// TIA Portal project "labE000120203ICA" (V15.1)

(* hardware
DEVICE "S7300/ET200M station_2"  S7-300 station
   slot 0: "Rail_0"  Rail  6ES7 390-1***0-0AA0
   slot 2: "PLC_Shaft"  CPU 314C-2 PN/DP  6ES7 314-6EH04-0AB0  V3.3
      slot 2: "PROFINET interface_1"  PN-IO
         slot 1: "Port_1"  Port
         slot 2: "Port_2"  Port
      slot 5: "DI 24/DO 16_1"  DI24/DO16
      slot 6: "AI 5/AO 2_1"  AI5/AO2
      slot 7: "Count_1"  Counter
      slot 8: "Positioning_1"  Positioning
DEVICE "HMI_Shaft"  KTP700 Basic PN
   slot 0: "HMI_Shaft"  KTP700 Basic PN  6AV2 123-2GB03-0AX0  15.1.0.0
   slot 1: "HMI_RT_2"  KTP700 Basic PN  6AV2 123-2GB03-0AX0  15.1.0.0
   slot 5: "HMI_Shaft.IE_CP_1"  PROFINET Interface  15.0.1.0
      slot 1: "PROFINET Interface_1"  PROFINET Interface
         slot 1: "Port_1"  Port
DEVICE "ET 200SP station_1"  ET 200SP-Station
   slot 0: "Rack_0"  Rack  6ES5 710-8MAx1
   slot 0: "IO device_1"  IM 155-6 PN/2 HF  6ES7 155-6AU01-0CN0  V4.2
   slot 1: "Server module_1"  Server module  6ES7 193-6PA00-0AA0  V1.1
      slot 1: "Server module_1"  Server module
   slot 127: "BA 2xRJ45"  BA 2xRJ45  6ES7 193-6AR00-0AA0  V0.0
      slot 1: "Port_1"  X1 P1 R  6ES7 193-6AR00-0AA0  V0.0
      slot 2: "Port_2"  X1 P2 R  6ES7 193-6AR00-0AA0  V0.0
DEVICE "S71500/ET200MP station_1"  S7-1500 station
   slot 0: "Rail_0"  Rack  6ES7 590-1***0-0AA0
   slot 1: "PLC_1"  CPU 1516-3 PN/DP  6ES7 516-3AN01-0AB0  V2.6
      slot 3: "CPU display_1"  6ES7591-1BA00-0AA0
*)

// ===== PLC "PLC_Shaft"  CPU 314C-2 PN/DP =====

TYPE "carousel"
   STRUCT
      carousel : Array[0..7] of Int;
   END_STRUCT;
END_TYPE

TYPE "Sequence"
VERSION : 0.1
   STRUCT
      actual : "step";
      old : "step";
      break : "step";
   END_STRUCT;
END_TYPE

TYPE "step"
VERSION : 0.1
   STRUCT
      "step" : Array[0..25] of Bool;
   END_STRUCT;
END_TYPE

TYPE "CTRL"
VERSION : 0.1
   STRUCT
      emergency_stop : Bool;
      trigger : Bool;
      trigger_flank : Bool;
      trigger_toggle : Bool;
      trigger_hulp : Bool;
      enable_step : Bool;
      auto : Bool;
      onestep : Bool;
      step_stop : Bool;
      step_break : Bool;
      toggle_hulp : Bool;
      break_on : Bool;
   END_STRUCT;
END_TYPE

TYPE "grafcet_data"
VERSION : 0.1
   STRUCT
      MyCTRL : "CTRL";
      Mygrafcet : "Sequence";
   END_STRUCT;
END_TYPE

DATA_BLOCK "Tafel_As_DB"   // DB1
{ S7_Optimized_Access := 'FALSE' }
VERSION : 0.1
// stored: InstanceOfName Tafel_As
"Tafel_As"
BEGIN
END_DATA_BLOCK

FUNCTION_BLOCK "Tafel_As"   // FB1, SCL
{ S7_Optimized_Access := 'FALSE' }
VERSION : 0.1
   VAR_INPUT
      sensorA0 : Bool;
      sensorA1 : Bool;
      sensorB0 : Bool;
      sensorB1 : Bool;
      sensorC0 : Bool;
      sensorC1 : Bool;
      sensorD0 : Bool;
      sensorD1 : Bool;
      sensorF1 : Bool;
      sensorG0 : Bool;
      sensorG1 : Bool;
      sensorV1 : Bool;
      sensorV2 : Bool;
      sensorDm : Bool;
      sensorDp : Bool;
      sensorJ0 : Bool;
   END_VAR
   VAR_OUTPUT
      "CilA+" : Bool;
      "CilB+" : Bool;
      "CilC+" : Bool;
      "CilC-" : Bool;
      "CilD+" : Bool;
      "CilE+" : Bool;
      "CilF+" : Bool;
      "CilG+" : Bool;
      "CilH+" : Bool;
      "CilI+" : Bool;
      "CilK+" : Bool;
      "CilJ+" : Bool;
      "ZV1+" : Bool;
      "ZV2+" : Bool;
   END_VAR
   VAR
      "cilinderA+" : "cilinder";
      "cilinderB+" : "cilinder";
      "cilinderC+" : "cilinder";
      "cilinderC-" : "cilinder";
      "cilinderD+" : "cilinder";
      "cilinderE+" : "cilinder";
      "cilinderF+" : "cilinder";
      "cilinderG+" : "cilinder";
      "cilinderH+" : "cilinder";
      "cilinderI+" : "cilinder";
      "cilinderK+" : "cilinder";
      "cilinderJ+" : "cilinder";
      "zuigerV1+" : "cilinder";
      "zuigerV2+" : "cilinder";
      seq_as_einde_invoer : "grafcet_data";
      seq_as_draaien_invoer : "grafcet_data";
      seq_sorteringsarm_invoer : "grafcet_data";
      seq_detectiesensoren_invoer : "grafcet_data";
      seq_carousel_invoer : "grafcet_data";
      timer300ms : TON;
   END_VAR
BEGIN
   REGION Aanmaken grafcets
       // Statement section REGION
       "ctrl_seq"(size := 10,
                  sequences := #seq_as_einde_invoer);

       "ctrl_seq"(size := 10,
                  sequences := #seq_as_draaien_invoer);

       "ctrl_seq"(size := 10,
                  sequences := #seq_sorteringsarm_invoer);

       "ctrl_seq"(size := 10,
                  sequences := #seq_detectiesensoren_invoer);

       "ctrl_seq"(size := 10,
                  sequences := #seq_carousel_invoer);
   END_REGION


   REGION Stappen grafcet as plaatsen op lager
       // Statement section REGION
       "Seq1-->1"(actualstep := 1,
                  nextstep := 2,
                  condition := #sensorB0,
                  Sequence := #seq_as_einde_invoer);

       "Seq1-->1"(actualstep := 2,
                  nextstep := 3,
                  condition := #sensorA0,
                  Sequence := #seq_as_einde_invoer);

       "Seq1-->1"(actualstep := 3,
                  nextstep := 4,
                  condition := #sensorA1,
                  Sequence := #seq_as_einde_invoer);

       "Seq1-->1"(actualstep := 4,
                  nextstep := 5,
                  condition := #sensorV1,
                  Sequence := #seq_as_einde_invoer);

       "Seq1-->1"(actualstep := 5,
                  nextstep := 6,
                  condition := #sensorA0,
                  Sequence := #seq_as_einde_invoer);

       "Seq1-->1"(actualstep := 6,
                  nextstep := 7,
                  condition := #sensorB1,
                  Sequence := #seq_as_einde_invoer);

       "Seq1-->1"(actualstep := 7,
                  nextstep := 8,
                  condition := #sensorA1,
                  Sequence := #seq_as_einde_invoer);

       "Seq1-->1"(actualstep := 8,
                  nextstep := 9,
                  condition := #timer300ms.Q,
                  Sequence := #seq_as_einde_invoer);

       "Seq1-->1"(actualstep := 9,
                  nextstep := 1,
                  condition := #sensorA0,
                  Sequence := #seq_as_einde_invoer);
   END_REGION

   REGION Stappen grafcet as draaien
       // Statement section REGION
       "Seq1-->1"(actualstep := 1,
                  nextstep := 2,
                  condition := #sensorG0,
                  Sequence := #seq_as_draaien_invoer);

       "Seq1-->1"(actualstep := 2,
                  nextstep := 3,
                  condition := #sensorG1,
                  Sequence := #seq_as_draaien_invoer);

       "Seq1-->1"(actualstep := 3,
                  nextstep := 4,
                  condition := #timer300ms.Q,
                  Sequence := #seq_as_draaien_invoer);

       "Seq1-->1"(actualstep := 4,
                  nextstep := 5,
                  condition := #sensorG0,
                  Sequence := #seq_as_draaien_invoer);

       "Seq1-->1"(actualstep := 5,
                  nextstep := 6,
                  condition := #timer300ms.Q,
                  Sequence := #seq_as_draaien_invoer);

       "Seq1-->1"(actualstep := 6,
                  nextstep := 7,
                  condition := #sensorG1,
                  Sequence := #seq_as_draaien_invoer);

       "Seq1-->1"(actualstep := 7,
                  nextstep := 8,
                  condition := #sensorG1,
                  Sequence := #seq_as_draaien_invoer);

       "Seq1-->1"(actualstep := 8,
                  nextstep := 1,
                  condition := #timer300ms.Q,
                  Sequence := #seq_as_draaien_invoer);
   END_REGION

   REGION Stappen grafset sorteringsarm
       // Statement section REGION
       "Seq1-->1"(actualstep := 1,
                  nextstep := 2,
                  condition := #sensorC0,
                  Sequence := #seq_sorteringsarm_invoer);

       "Seq1-->1"(actualstep := 2,
                  nextstep := 3,
                  condition := #sensorC1,
                  Sequence := #seq_sorteringsarm_invoer);

       "Seq1-->1"(actualstep := 3,
                  nextstep := 4,
                  condition := #sensorD1,
                  Sequence := #seq_sorteringsarm_invoer);

       "Seq1-->1"(actualstep := 4,
                  nextstep := 5,
                  condition := #sensorV2,
                  Sequence := #seq_sorteringsarm_invoer);

       "Seq1-->1"(actualstep := 5,
                  nextstep := 1,
                  condition := #sensorD0,
                  Sequence := #seq_sorteringsarm_invoer);
   END_REGION

   REGION Stappen grafcet carousel
       // Statement section REGION
       "Seq1-->1"(actualstep:=1,
                  nextstep:=2,
                  condition:=#sensorJ0,
                  Sequence:=#seq_carousel_invoer);

       "Seq1-->1"(actualstep:=2,
                  nextstep:=3,
                  condition:=#seq_as_draaien_invoer.Mygrafcet.actual.step[8] AND #seq_as_einde_invoer.Mygrafcet.actual.step[9] AND #seq_sorteringsarm_invoer.Mygrafcet.actual.step[5],
                  Sequence:=#seq_carousel_invoer);

       "Seq1-->1"(actualstep:=3,
                  nextstep:=4,
                  condition:=#timer300ms.Q,
                  Sequence:=#seq_carousel_invoer);

       "Seq1-->1"(actualstep:=4,
                  nextstep:=5,
                  condition:=#timer300ms.Q AND #sensorJ0 = FALSE,
                  Sequence:=#seq_carousel_invoer);

       "Seq1-->1"(actualstep:=5,
                  nextstep:=1,
                  condition:=#timer300ms.Q,
                  Sequence:=#seq_carousel_invoer);

   END_REGION



   REGION Uitgangen as draaien
       // Statement section REGION
       #"cilinderH+"(manueelinschuiven := false,
                     manueeluitschuiven := false,
                     AutomatischUitschuiven := #seq_as_draaien_invoer.Mygrafcet.actual.step[4] OR #seq_as_einde_invoer.Mygrafcet.actual.step[5] OR #seq_as_einde_invoer.Mygrafcet.actual.step[6] OR #seq_as_einde_invoer.Mygrafcet.actual.step[7],
                     ManAuto := false,
                     "IL uitschuiven" := false,
                     "IL inschuiven" := false,
                     "Eindeloop In" := false,
                     "Eindeloop Uit" := false,
                     "Reset Foutmelding" := false,
                     TeachMode := false,
                     MargeLooptijden := T#0ms,
                     "Max Aantal slagen" := 0,
                     "Reset Onderhoud" := false,
                     Noodstop := false,
                     AansturingMono =>#"CilH+");

       #"cilinderG+"(manueelinschuiven := false,
                     manueeluitschuiven := false,
                     AutomatischUitschuiven:=#seq_as_draaien_invoer.Mygrafcet.actual.step[1] OR #seq_as_draaien_invoer.Mygrafcet.actual.step[2] OR #seq_as_draaien_invoer.Mygrafcet.actual.step[5] OR #seq_as_draaien_invoer.Mygrafcet.actual.step[6],
                     ManAuto := false,
                     "IL uitschuiven" := false,
                     "IL inschuiven" := false,
                     "Eindeloop In" := false,
                     "Eindeloop Uit" := false,
                     "Reset Foutmelding" := false,
                     TeachMode := false,
                     MargeLooptijden := T#0ms,
                     "Max Aantal slagen" := 0,
                     "Reset Onderhoud" := false,
                     Noodstop := false,
                     AansturingMono=>#"CilG+");

       #"cilinderI+"(manueelinschuiven := false,
                     manueeluitschuiven := false,
                     AutomatischUitschuiven:=#seq_as_draaien_invoer.Mygrafcet.actual.step[2] OR #seq_as_draaien_invoer.Mygrafcet.actual.step[3] OR #seq_as_draaien_invoer.Mygrafcet.actual.step[4] OR #seq_as_draaien_invoer.Mygrafcet.actual.step[5],
                     ManAuto := false,
                     "IL uitschuiven" := false,
                     "IL inschuiven" := false,
                     "Eindeloop In" := false,
                     "Eindeloop Uit" := false,
                     "Reset Foutmelding" := false,
                     TeachMode := false,
                     MargeLooptijden := T#0ms,
                     "Max Aantal slagen" := 0,
                     "Reset Onderhoud" := false,
                     Noodstop := false,
                     AansturingMono=>#"CilI+");

   END_REGION

   REGION Uitgangen as plaatsen op lager
       // Statement section REGION
       #"cilinderA+"(manueelinschuiven := false,
                     manueeluitschuiven := false,
                     AutomatischUitschuiven := #seq_as_einde_invoer.Mygrafcet.actual.step[2] OR #seq_as_einde_invoer.Mygrafcet.actual.step[3] OR #seq_as_einde_invoer.Mygrafcet.actual.step[6] OR #seq_as_einde_invoer.Mygrafcet.actual.step[7],
                     ManAuto := false,
                     "IL uitschuiven" := #sensorA0,
                     "IL inschuiven" := #sensorA1,
                     "Eindeloop In" := false,
                     "Eindeloop Uit" := false,
                     "Reset Foutmelding" := false,
                     TeachMode := false,
                     MargeLooptijden := T#0ms,
                     "Max Aantal slagen" := 0,
                     "Reset Onderhoud" := false,
                     Noodstop := false,
                     AansturingMono => #"CilA+");


       #"cilinderB+"(manueelinschuiven := false,
                     manueeluitschuiven := false,
                     AutomatischUitschuiven := #seq_as_einde_invoer.Mygrafcet.actual.step[5] OR #seq_as_einde_invoer.Mygrafcet.actual.step[6] OR #seq_as_einde_invoer.Mygrafcet.actual.step[7] OR #seq_as_einde_invoer.Mygrafcet.actual.step[8],
                     ManAuto := false,
                     "IL uitschuiven" := #sensorB0,
                     "IL inschuiven" := #sensorB1,
                     "Eindeloop In" := false,
                     "Eindeloop Uit" := false,
                     "Reset Foutmelding" := false,
                     TeachMode := false,
                     MargeLooptijden := T#0ms,
                     "Max Aantal slagen" := 0,
                     "Reset Onderhoud" := false,
                     Noodstop := false,
                     AansturingMono => #"CilB+");


       #"zuigerV1+"(manueelinschuiven := false,
                    manueeluitschuiven := false,
                    AutomatischUitschuiven:=#seq_as_einde_invoer.Mygrafcet.actual.step[3] OR #seq_as_einde_invoer.Mygrafcet.actual.step[4] OR #seq_as_einde_invoer.Mygrafcet.actual.step[5] OR #seq_as_einde_invoer.Mygrafcet.actual.step[6],
                    ManAuto := false,
                    "IL uitschuiven" := false,
                    "IL inschuiven" := false,
                    "Eindeloop In" := false,
                    "Eindeloop Uit" := false,
                    "Reset Foutmelding" := false,
                    TeachMode := false,
                    MargeLooptijden := T#0ms,
                    "Max Aantal slagen" := 0,
                    "Reset Onderhoud" := false,
                    Noodstop := false,
                    AansturingMono=>#"ZV1+");
   END_REGION

   REGION Uitgangen sorteringsarm
       // Statement section REGION
       #"cilinderC+"(manueelinschuiven := false,
                     manueeluitschuiven := false,
                     AutomatischUitschuiven:=#seq_sorteringsarm_invoer.Mygrafcet.actual.step[1],
                     ManAuto := false,
                     "IL uitschuiven" := false,
                     "IL inschuiven" := false,
                     "Eindeloop In" := false,
                     "Eindeloop Uit" := false,
                     "Reset Foutmelding" := false,
                     TeachMode := false,
                     MargeLooptijden := T#0ms,
                     "Max Aantal slagen" := 0,
                     "Reset Onderhoud" := false,
                     Noodstop := false,
                     AansturingMono=>#"CilC+");

       #"cilinderC-"(manueelinschuiven := false,
                     manueeluitschuiven := false,
                     AutomatischUitschuiven:=#seq_sorteringsarm_invoer.Mygrafcet.actual.step[5],
                     ManAuto := false,
                     "IL uitschuiven" := false,
                     "IL inschuiven" := false,
                     "Eindeloop In" := false,
                     "Eindeloop Uit" := false,
                     "Reset Foutmelding" := false,
                     TeachMode := false,
                     MargeLooptijden := T#0ms,
                     "Max Aantal slagen" := 0,
                     "Reset Onderhoud" := false,
                     Noodstop := false,
                     AansturingMono=>#"CilC-");

       #"cilinderD+"(manueelinschuiven := false,
                     manueeluitschuiven := false,
                     AutomatischUitschuiven:=#seq_sorteringsarm_invoer.Mygrafcet.actual.step[2] OR #seq_sorteringsarm_invoer.Mygrafcet.actual.step[3],
                     ManAuto := false,
                     "IL uitschuiven" := false,
                     "IL inschuiven" := false,
                     "Eindeloop In" := false,
                     "Eindeloop Uit" := false,
                     "Reset Foutmelding" := false,
                     TeachMode := false,
                     MargeLooptijden := T#0ms,
                     "Max Aantal slagen" := 0,
                     "Reset Onderhoud" := false,
                     Noodstop := false,
                     AansturingMono=>#"CilD+");

       #"zuigerV2+"(manueelinschuiven := false,
                    manueeluitschuiven := false,
                    AutomatischUitschuiven:=#seq_sorteringsarm_invoer.Mygrafcet.actual.step[3] OR #seq_sorteringsarm_invoer.Mygrafcet.actual.step[4] OR #seq_sorteringsarm_invoer.Mygrafcet.actual.step[5],
                    ManAuto := false,
                    "IL uitschuiven" := false,
                    "IL inschuiven" := false,
                    "Eindeloop In" := false,
                    "Eindeloop Uit" := false,
                    "Reset Foutmelding" := false,
                    TeachMode := false,
                    MargeLooptijden := T#0ms,
                    "Max Aantal slagen" := 0,
                    "Reset Onderhoud" := false,
                    Noodstop := false,
                    AansturingMono=>#"ZV2+");

   END_REGION

   REGION Uitgang carousel
       // Statement section REGION
       #"cilinderK+"(manueelinschuiven := false,
                     manueeluitschuiven := false,
                     AutomatischUitschuiven:=#seq_carousel_invoer.Mygrafcet.actual.step[2] OR #seq_carousel_invoer.Mygrafcet.actual.step[3],
                     ManAuto := false,
                     "IL uitschuiven" := false,
                     "IL inschuiven" := false,
                     "Eindeloop In" := false,
                     "Eindeloop Uit" := false,
                     "Reset Foutmelding" := false,
                     TeachMode := false,
                     MargeLooptijden := T#0ms,
                     "Max Aantal slagen" := 0,
                     "Reset Onderhoud" := false,
                     Noodstop := false,
                     AansturingMono=>#"CilK+");

       #"cilinderJ+"(manueelinschuiven := false,
                     manueeluitschuiven := false,
                     AutomatischUitschuiven:=#seq_carousel_invoer.Mygrafcet.actual.step[3] OR #seq_carousel_invoer.Mygrafcet.actual.step[4],
                     ManAuto := false,
                     "IL uitschuiven" := false,
                     "IL inschuiven" := false,
                     "Eindeloop In" := false,
                     "Eindeloop Uit" := false,
                     "Reset Foutmelding" := false,
                     TeachMode := false,
                     MargeLooptijden := T#0ms,
                     "Max Aantal slagen" := 0,
                     "Reset Onderhoud" := false,
                     Noodstop := false,
                     AansturingMono=>#"CilJ+");

   END_REGION



   #timer300ms(IN := #seq_carousel_invoer.Mygrafcet.actual.step[2] OR #seq_carousel_invoer.Mygrafcet.actual.step[3] OR #seq_carousel_invoer.Mygrafcet.actual.step[4] OR #seq_as_einde_invoer.Mygrafcet.actual.step[7] OR #seq_as_draaien_invoer.Mygrafcet.actual.step[3] OR #seq_as_draaien_invoer.Mygrafcet.actual.step[5] OR #seq_as_draaien_invoer.Mygrafcet.actual.step[7],
               PT := t#300ms);
END_FUNCTION_BLOCK

ORGANIZATION_BLOCK "Main"   // OB1, LAD
TITLE = "Main Program Sweep (Cycle)"
{ S7_Optimized_Access := 'FALSE' }
VERSION : 0.1
   VAR_TEMP
      OB1_EV_CLASS : Byte;   // Bits 0-3 = 1 (Coming event), Bits 4-7 = 1 (Event class 1)
      OB1_SCAN_1 : Byte;   // 1 (Cold restart scan 1 of OB 1), 3 (Scan 2-n of OB 1)
      OB1_PRIORITY : Byte;   // Priority of OB Execution
      OB1_OB_NUMBR : Byte;   // 1 (Organization block 1, OB1)
      OB1_RESERVED_1 : Byte;   // Reserved for system
      OB1_RESERVED_2 : Byte;   // Reserved for system
      OB1_PREV_CYCLE : Int;   // Cycle time of previous OB1 scan (milliseconds)
      OB1_MIN_CYCLE : Int;   // Minimum cycle time of OB1 (milliseconds)
      OB1_MAX_CYCLE : Int;   // Maximum cycle time of OB1 (milliseconds)
      OB1_DATE_TIME : Date_And_Time;   // Date and time OB1 started
   END_VAR
BEGIN

REGION Network 1
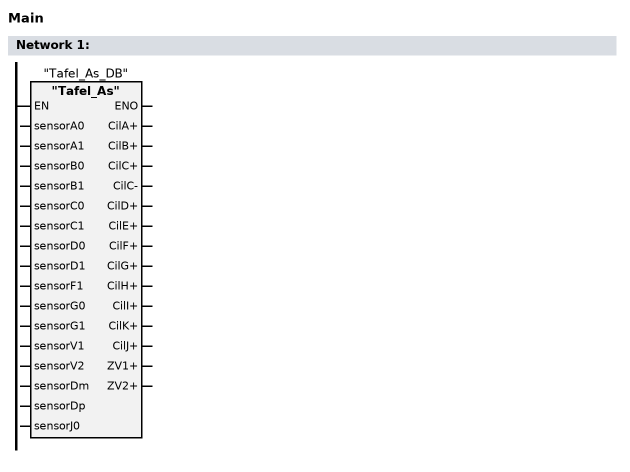
   RUNG wire#powerrail
      "Tafel_As_DB"(sensorA0 :=, sensorA1 :=, sensorB0 :=, sensorB1 :=, sensorC0 :=, sensorC1 :=, sensorD0 :=, sensorD1 :=, sensorF1 :=, sensorG0 :=, sensorG1 :=, sensorV1 :=, sensorV2 :=, sensorDm :=, sensorDp :=, sensorJ0 :=, "CilA+" =>, "CilB+" =>, "CilC+" =>, "CilC-" =>, "CilD+" =>, "CilE+" =>, "CilF+" =>, "CilG+" =>, "CilH+" =>, "CilI+" =>, "CilK+" =>, "CilJ+" =>, "ZV1+" =>, "ZV2+" =>)
   END_RUNG
   // the same network as SCL:
   "Tafel_As_DB"();   // "Tafel_As"
END_REGION
END_ORGANIZATION_BLOCK

ORGANIZATION_BLOCK "COMPLETE RESTART"   // OB100, SCL
TITLE = "Complete Restart"
{ S7_Optimized_Access := 'FALSE' }
VERSION : 0.1
   VAR_TEMP
      OB100_EV_CLASS : Byte;   // 16#13, Event class 1, Entering event state, Event logged in diagnostic buffer
      OB100_STRTUP : Byte;   // 16#81/82/83/84 Method of startup
      OB100_PRIORITY : Byte;   // Priority of OB Execution
      OB100_OB_NUMBR : Byte;   // 100 (Organization block 100, OB100)
      OB100_RESERVED_1 : Byte;   // Reserved for system
      OB100_RESERVED_2 : Byte;   // Reserved for system
      OB100_STOP : Word;   // Event that caused CPU to stop (16#4xxx)
      OB100_STRT_INFO : DWord;   // Information on how system started
      OB100_DATE_TIME : Date_And_Time;   // Date and time OB100 started
   END_VAR
BEGIN
   "initialisation"(number:=20,
                    Normal_sequence:="Mijn_Tafel_Lager".seq_invoer);
   "initialisation"(number := 20,
                    Normal_sequence := "Mijn_Tafel_Lager".seq_uitvoer);
END_ORGANIZATION_BLOCK

// folder: basisclasses

FUNCTION_BLOCK "cilinder"   // FB8, FBD
{ S7_Optimized_Access := 'FALSE' }
VERSION : 0.1
   VAR_INPUT
      manueelinschuiven : Bool;
      manueeluitschuiven : Bool;   // '1' betekent uitschuiven '0' inschuiven
      AutomatischUitschuiven : Bool;
      ManAuto : Bool;   // '1' betekent Manueel '0' Automatisch
      "IL uitschuiven" : Bool;   // '1' betekent vergrendeld
      "IL inschuiven" : Bool;   // '1' betekent vergrendeld
      "Eindeloop In" : Bool;
      "Eindeloop Uit" : Bool;
      "Reset Foutmelding" : Bool;
      TeachMode : Bool;   // '1' wanneer er tijden worden ingesteld
      MargeLooptijden : Time;   // marge instellen looptijdbewaking
      "Max Aantal slagen" : Int;   // Aantal slagen voor onderhoud
      "Reset Onderhoud" : Bool;
      Noodstop : Bool;   // '0' betekent noodstop actief
   END_VAR
   VAR_OUTPUT
      AansturingMono : Bool;
      AansturingAanBist : Bool;
      AansturingUitBist : Bool;
      "Alarm Looptijd" : Bool;   // Te lang om dicht of open te schuiven
      "Alarm Interlock" : Bool;   // poging om te bedienen bij aanwezige interlock
      "Alarm Noodstop" : Bool;
      "Alarm Eindeloop" : Bool;   // wanneer elektrisch probleem op eindelopen
      "Alarm Onderhoud" : Bool;
   END_VAR
   VAR
      grafcetssturing : Bool;
      "Referentie Looptijd Inschuiven" : Time;
      "Referentie Looptijd Uitschuiven" : Time;
      "Werkelijke Looptijd Inschuiven" : Time;
      "Werkelijke Looptijd Uitschuiven" : Time;
      "Werkelijke Aantal Slagen" : Int;
      OnderhoudTeller : CTD;
      SROnderhoud : Bool;
      SREindeloop : Bool;
      SRNoodstop : Bool;
      FlankManUit : Bool;
      FlankAutoUit : Bool;
      SRInterlock : Bool;
      FlankManIN : Bool;
      FlankAutoIN : Bool;
      TeachTimer : TON;
      FlankEindeUit : Bool;
      FlankEindeIn : Bool;
      RefTijdIn : Int;
      RefTijdUit : Int;
      WerkTijdIn : Int;
      WerkTijdUit : Int;
      SRLooptijd : Bool;
      FlankEindeUit1 : Bool;
      FlankEindeIn1 : Bool;
      eindeloopuitflank : Bool;
      eindeloopinflank : Bool;
      bewaaktijdeninschuiven : "bewaaktijden";
      bewaaktijdenuitschuif : "bewaaktijden";
      flankmanueelinschuiven : Bool;
      flankmanueeluitschuiven : Bool;
      movesetreset : Bool;
      PercentageSlagen : Real;
      Real_aantal : Real;
      Monosturing : Bool;
      BisturingAan : Bool;
      BisturingUit : Bool;
      FposAansturing : Bool;
      FnegAansturing : Bool;
      DINT_aantal : DInt;
   END_VAR
   VAR_TEMP
      ondergrensin : Int;
      bovengrensuit : Int;
      ondergrensuit : Int;
      vals : Bool;
      bovengrensin : Int;
   END_VAR
   VAR_TEMP   // added for the SCL form of the ladder/FBD networks
      _w1 : Bool;
      _w2 : Bool;
      _w3 : Bool;
      _w4 : Bool;
      _w5 : Bool;
   END_VAR
BEGIN

REGION Network 1: Onderhoud
   // Teller van de cilindir om na x aantal slagen onderhoud uit te voeren op de cilindir.
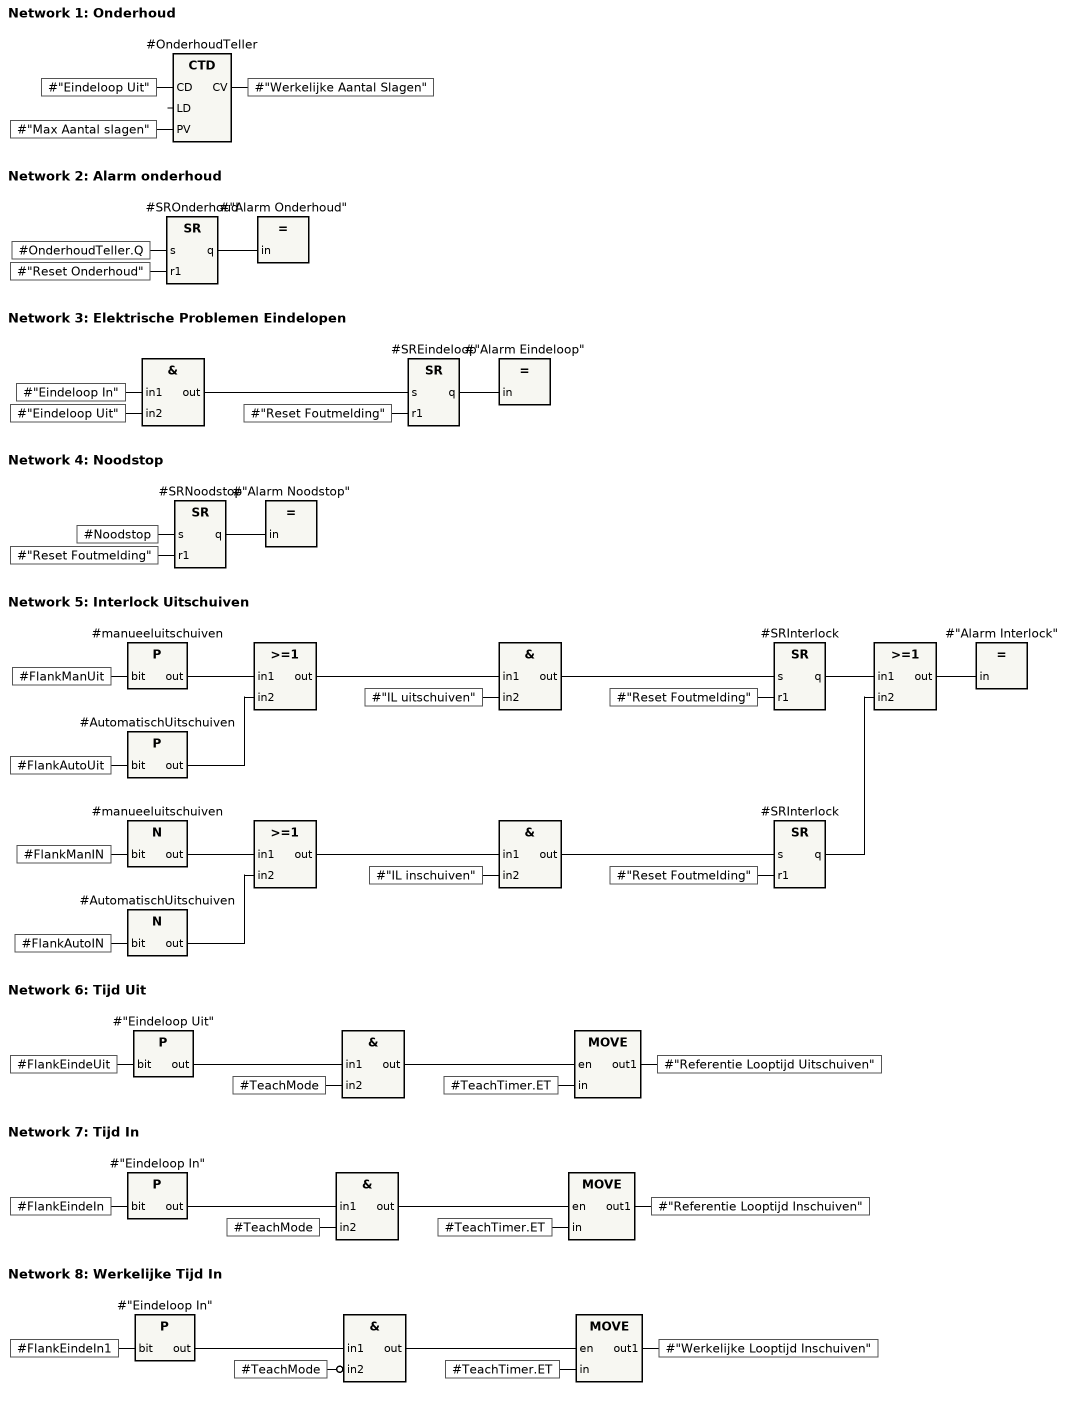
   #OnderhoudTeller.CTD(CD := #"Eindeloop Uit", PV := #"Max Aantal slagen", CV => #"Werkelijke Aantal Slagen");
END_REGION

REGION Network 2: Alarm onderhoud
   // Weergave van wanneer de teller zijn aantal slagen heeft bereikt, kan gereset worden
   IF #OnderhoudTeller.Q THEN
       #SROnderhoud := TRUE;   // SR flip-flop
   END_IF;
   IF #"Reset Onderhoud" THEN #SROnderhoud := FALSE; END_IF;
   #"Alarm Onderhoud" := #SROnderhoud;
END_REGION

REGION Network 3: Elektrische Problemen Eindelopen
   // Beide eindelopen mogen nooit beide aanliggen, dit is fysisch niet mogelijk en is dus een elektrisch probleem
   IF #"Eindeloop In" AND #"Eindeloop Uit" THEN
       #SREindeloop := TRUE;   // SR flip-flop
   END_IF;
   IF #"Reset Foutmelding" THEN #SREindeloop := FALSE; END_IF;
   #"Alarm Eindeloop" := #SREindeloop;
END_REGION

REGION Network 4: Noodstop
   // de fysishe noodstop is nc contact
   IF #Noodstop THEN
       #SRNoodstop := TRUE;   // SR flip-flop
   END_IF;
   IF #"Reset Foutmelding" THEN #SRNoodstop := FALSE; END_IF;
   #"Alarm Noodstop" := #SRNoodstop;
END_REGION

REGION Network 5: Interlock Uitschuiven
   // Alarm voor wanneer de cilindir wordt aangestuurd maar de interlock is actief.
   #_w1 := #manueeluitschuiven AND NOT #FlankManUit;   // rising edge of #manueeluitschuiven
   #FlankManUit := #manueeluitschuiven;
   #_w2 := #AutomatischUitschuiven AND NOT #FlankAutoUit;   // rising edge of #AutomatischUitschuiven
   #FlankAutoUit := #AutomatischUitschuiven;
   IF (#_w1 OR #_w2) AND #"IL uitschuiven" THEN
       #SRInterlock := TRUE;   // SR flip-flop
   END_IF;
   IF #"Reset Foutmelding" THEN #SRInterlock := FALSE; END_IF;
   #_w3 := NOT #manueeluitschuiven AND #FlankManIN;   // falling edge of #manueeluitschuiven
   #FlankManIN := #manueeluitschuiven;
   #_w4 := NOT #AutomatischUitschuiven AND #FlankAutoIN;   // falling edge of #AutomatischUitschuiven
   #FlankAutoIN := #AutomatischUitschuiven;
   #_w5 := #SRInterlock;
   IF (#_w3 OR #_w4) AND #"IL inschuiven" THEN
       #SRInterlock := TRUE;   // SR flip-flop
   END_IF;
   IF #"Reset Foutmelding" THEN #SRInterlock := FALSE; END_IF;
   #"Alarm Interlock" := #_w5 OR #SRInterlock;
END_REGION

REGION Network 6: Tijd Uit
   // cilinder in teach mode vastleggen referentietijd uitschuiven
   #_w1 := #"Eindeloop Uit" AND NOT #FlankEindeUit;   // rising edge of #"Eindeloop Uit"
   #FlankEindeUit := #"Eindeloop Uit";
   IF #_w1 AND #TeachMode THEN #"Referentie Looptijd Uitschuiven" := #TeachTimer.ET; END_IF;
END_REGION

REGION Network 7: Tijd In
   // cilinder in teach mode vastleggen referentietijd inschuiven
   #_w1 := #"Eindeloop In" AND NOT #FlankEindeIn;   // rising edge of #"Eindeloop In"
   #FlankEindeIn := #"Eindeloop In";
   IF #_w1 AND #TeachMode THEN #"Referentie Looptijd Inschuiven" := #TeachTimer.ET; END_IF;
END_REGION

REGION Network 8: Werkelijke Tijd In
   // cilinder niet in teach mode vastleggen werkelijke tijd inschuiven
   #_w1 := #"Eindeloop In" AND NOT #FlankEindeIn1;   // rising edge of #"Eindeloop In"
   #FlankEindeIn1 := #"Eindeloop In";
   IF #_w1 AND NOT #TeachMode THEN #"Werkelijke Looptijd Inschuiven" := #TeachTimer.ET; END_IF;
END_REGION

REGION Network 9: Werkelijke Tijd Uit
   // cilinder niet in teach mode vastleggen werkelijke tijd uitschuiven
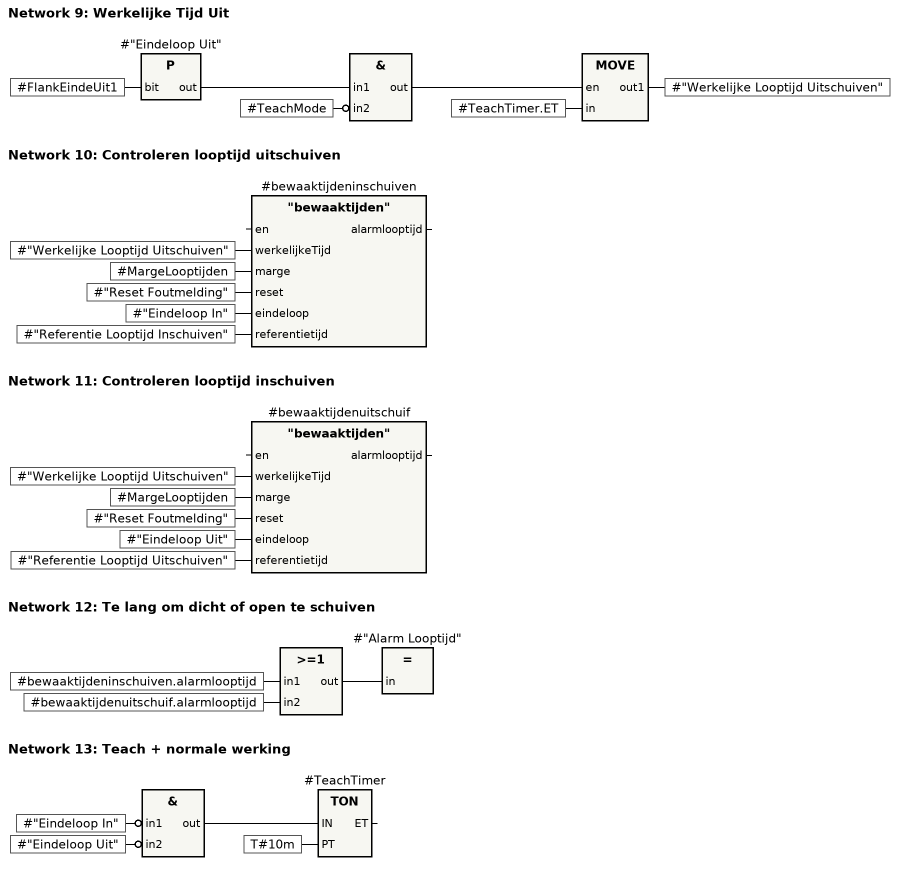
   #_w1 := #"Eindeloop Uit" AND NOT #FlankEindeUit1;   // rising edge of #"Eindeloop Uit"
   #FlankEindeUit1 := #"Eindeloop Uit";
   IF #_w1 AND NOT #TeachMode THEN #"Werkelijke Looptijd Uitschuiven" := #TeachTimer.ET; END_IF;
END_REGION

REGION Network 10: Controleren looptijd uitschuiven
   #bewaaktijdeninschuiven(werkelijkeTijd := #"Werkelijke Looptijd Uitschuiven",   // "bewaaktijden"
                           marge := #MargeLooptijden,
                           reset := #"Reset Foutmelding",
                           eindeloop := #"Eindeloop In",
                           referentietijd := #"Referentie Looptijd Inschuiven");
END_REGION

REGION Network 11: Controleren looptijd inschuiven
   #bewaaktijdenuitschuif(werkelijkeTijd := #"Werkelijke Looptijd Uitschuiven",   // "bewaaktijden"
                          marge := #MargeLooptijden,
                          reset := #"Reset Foutmelding",
                          eindeloop := #"Eindeloop Uit",
                          referentietijd := #"Referentie Looptijd Uitschuiven");
END_REGION

REGION Network 12: Te lang om dicht of open te schuiven
   #"Alarm Looptijd" := #bewaaktijdeninschuiven.alarmlooptijd OR #bewaaktijdenuitschuif.alarmlooptijd;
END_REGION

REGION Network 13: Teach + normale werking
   #TeachTimer.TON(IN := NOT #"Eindeloop In" AND NOT #"Eindeloop Uit", PT := T#10m);
END_REGION

REGION Network 14: Sturen van de cilinder monostabiel
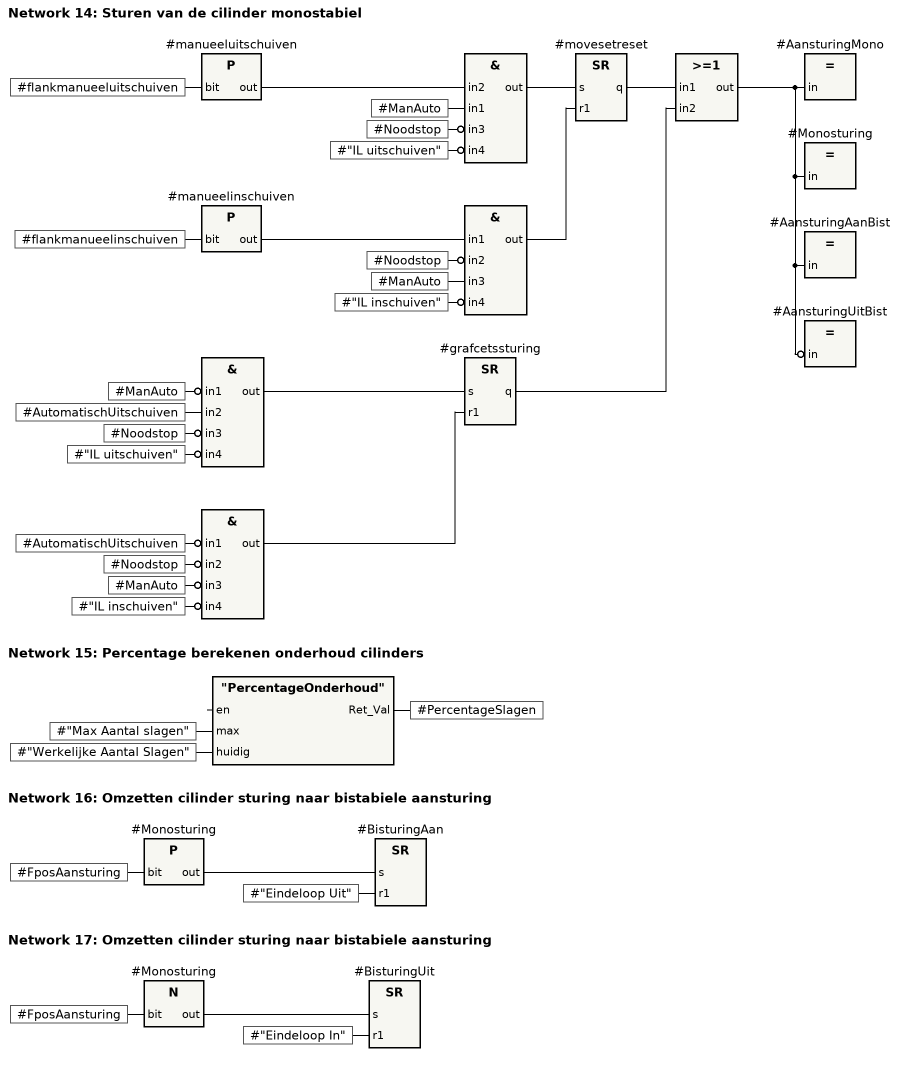
   #_w1 := #manueeluitschuiven AND NOT #flankmanueeluitschuiven;   // rising edge of #manueeluitschuiven
   #flankmanueeluitschuiven := #manueeluitschuiven;
   #_w2 := #manueelinschuiven AND NOT #flankmanueelinschuiven;   // rising edge of #manueelinschuiven
   #flankmanueelinschuiven := #manueelinschuiven;
   IF #_w1 AND #ManAuto AND NOT #Noodstop AND NOT #"IL uitschuiven" THEN
       #movesetreset := TRUE;   // SR flip-flop
   END_IF;
   IF #_w2 AND NOT #Noodstop AND #ManAuto AND NOT #"IL inschuiven" THEN #movesetreset := FALSE; END_IF;
   IF NOT #ManAuto AND #AutomatischUitschuiven AND NOT #Noodstop AND NOT #"IL uitschuiven" THEN
       #grafcetssturing := TRUE;   // SR flip-flop
   END_IF;
   IF NOT #AutomatischUitschuiven AND NOT #Noodstop AND NOT #ManAuto AND NOT #"IL inschuiven" THEN
       #grafcetssturing := FALSE;
   END_IF;
   #AansturingMono := #movesetreset OR #grafcetssturing;
   #Monosturing := #AansturingMono;
   #AansturingAanBist := #AansturingMono;
   #AansturingUitBist := NOT #AansturingMono;
END_REGION

REGION Network 15: Percentage berekenen onderhoud cilinders
   #PercentageSlagen := "PercentageOnderhoud"(max := #"Max Aantal slagen",
                           huidig := #"Werkelijke Aantal Slagen");
END_REGION

REGION Network 16: Omzetten cilinder sturing naar bistabiele aansturing
   #_w1 := #Monosturing AND NOT #FposAansturing;   // rising edge of #Monosturing
   #FposAansturing := #Monosturing;
   IF #_w1 THEN
       #BisturingAan := TRUE;   // SR flip-flop
   END_IF;
   IF #"Eindeloop Uit" THEN #BisturingAan := FALSE; END_IF;
END_REGION

REGION Network 17: Omzetten cilinder sturing naar bistabiele aansturing
   #_w1 := NOT #Monosturing AND #FposAansturing;   // falling edge of #Monosturing
   #FposAansturing := #Monosturing;
   IF #_w1 THEN
       #BisturingUit := TRUE;   // SR flip-flop
   END_IF;
   IF #"Eindeloop In" THEN #BisturingUit := FALSE; END_IF;
END_REGION
END_FUNCTION_BLOCK

FUNCTION_BLOCK "bewaaktijden"   // FB9, SCL
{ S7_Optimized_Access := 'FALSE' }
VERSION : 0.1
   VAR_INPUT
      werkelijkeTijd : Time;
      marge : Time;
      reset : Bool;
      eindeloop : Bool;
      referentietijd : Time;
   END_VAR
   VAR_OUTPUT
      alarmlooptijd : Bool;
   END_VAR
   VAR
      flankeindeloop : Bool;
   END_VAR
BEGIN
   IF ((#werkelijkeTijd > (#referentietijd + #marge)) OR (#werkelijkeTijd< (#referentietijd - #marge))) AND #eindeloop AND (NOT #flankeindeloop) THEN
       // Statement section IF
       #alarmlooptijd := TRUE;
   END_IF;
   IF #reset THEN
       // Statement section IF
       #alarmlooptijd := FALSE;
   END_IF;
   #flankeindeloop := #eindeloop;
END_FUNCTION_BLOCK

FUNCTION "PercentageOnderhoud" : Real   // FC2, SCL
{ S7_Optimized_Access := 'FALSE' }
VERSION : 0.1
   VAR_INPUT
      max : Int;
      huidig : Int;
   END_VAR
BEGIN
   #PercentageOnderhoud := INT_TO_REAL(#huidig) / INT_TO_REAL(#max) * 100;
END_FUNCTION

// folder: grafcet

FUNCTION "Seq1-->1" : Void   // FC1, SCL
{ S7_Optimized_Access := 'FALSE' }
VERSION : 0.1
   VAR_INPUT
      actualstep : Int;
      nextstep : Int;
      condition : Bool;
   END_VAR
   VAR_IN_OUT
      Sequence : "grafcet_data";
   END_VAR
BEGIN
   //Fonction permettant de passer d'une étape à une autre.


   IF #Sequence.Mygrafcet.old.step[#actualstep] AND #Sequence.MyCTRL.enable_step AND #condition THEN
       // Statement section IF
       #Sequence.Mygrafcet.actual.step[#nextstep] := true;
       #Sequence.Mygrafcet.actual.step[#actualstep] := false;

   END_IF;
END_FUNCTION

FUNCTION "Seq1-->2" : Void   // FC3, SCL
{ S7_Optimized_Access := 'FALSE' }
VERSION : 0.1
   VAR_INPUT
      actualstep : Int;
      nextstep1 : Int;
      nextstep2 : Int;
      condition : Bool;
   END_VAR
   VAR_IN_OUT
      Normal_Sequence : "grafcet_data";
   END_VAR
   VAR_TEMP
      VarConditon2 : Bool;
      VarConditon1 : Bool;
   END_VAR
BEGIN
   IF #Normal_Sequence.Mygrafcet.old.step[#actualstep] AND #Normal_Sequence.MyCTRL.enable_step AND #condition THEN
       // Statement section IF

       #Normal_Sequence.Mygrafcet.actual.step[#nextstep1] := true;
       #Normal_Sequence.Mygrafcet.actual.step[#nextstep2] := true;
       #Normal_Sequence.Mygrafcet.actual.step[#actualstep] := false;
       ;
   END_IF;
END_FUNCTION

FUNCTION "Seq2-->1" : Void   // FC4, SCL
{ S7_Optimized_Access := 'FALSE' }
VERSION : 0.1
   VAR_INPUT
      actualstep1 : Int;
      actualstep2 : Int;
      nextstep : Int;
      condition : Bool;
   END_VAR
   VAR_IN_OUT
      Normal_Sequence : "grafcet_data";
   END_VAR
BEGIN
   IF #Normal_Sequence.Mygrafcet.old.step[#actualstep1] AND #Normal_Sequence.Mygrafcet.old.step[#actualstep2] AND #Normal_Sequence.MyCTRL.enable_step AND #condition THEN
       // Statement section IF

       #Normal_Sequence.Mygrafcet.actual.step[#actualstep2] := FALSE;
       #Normal_Sequence.Mygrafcet.actual.step[#nextstep] := true;
       #Normal_Sequence.Mygrafcet.actual.step[#actualstep1] := false;
       ;
   END_IF;
END_FUNCTION

FUNCTION "Seq1--> END" : Void   // FC5, SCL
{ S7_Optimized_Access := 'FALSE' }
VERSION : 0.1
   VAR_INPUT
      actualstep : Int;
   END_VAR
   VAR_IN_OUT
      Sequence : "grafcet_data";
   END_VAR
BEGIN
   //Fonction permettant de passer d'une étape à une autre. Drain Step ( = missing next step)


   IF #Sequence.Mygrafcet.old.step[#actualstep] AND #Sequence.MyCTRL.enable_step THEN
       // Statement section IF    
       #Sequence.Mygrafcet.actual.step[#actualstep] := false;

   END_IF;
END_FUNCTION

FUNCTION "Grafcet_modus" : Void   // FC15, LAD
{ S7_Optimized_Access := 'FALSE' }
VERSION : 0.1
   VAR_IN_OUT
      ctrl : "CTRL";
   END_VAR
   VAR_TEMP   // added for the SCL form of the ladder/FBD networks
      _w1 : Bool;
   END_VAR
BEGIN

REGION Network 1
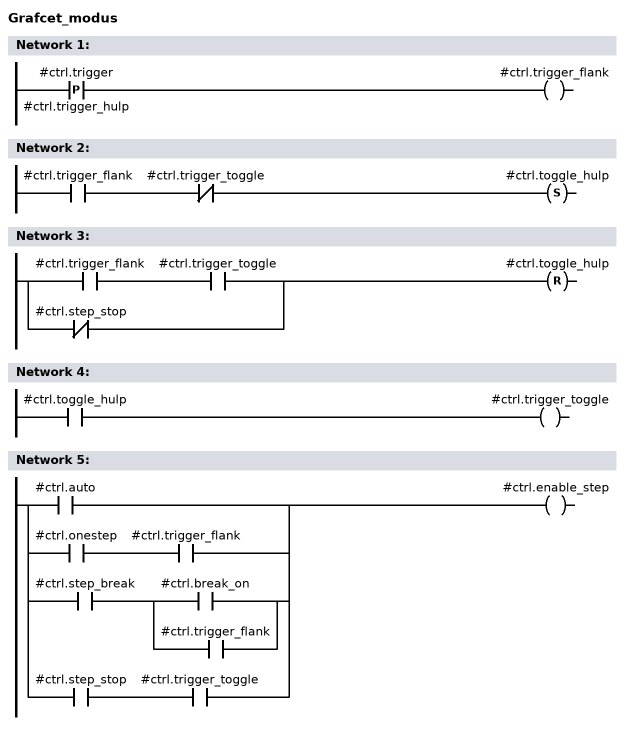
   RUNG wire#powerrail
      P_Contact(operand := #ctrl.trigger, bit := #ctrl.trigger_hulp)
      Coil( #ctrl.trigger_flank )
   END_RUNG
   // the same network as SCL:
   #_w1 := #ctrl.trigger AND NOT #ctrl.trigger_hulp;   // rising edge of #ctrl.trigger
   #ctrl.trigger_hulp := #ctrl.trigger;
   #ctrl.trigger_flank := #_w1;
END_REGION

REGION Network 2
   RUNG wire#powerrail
      Contact( #ctrl.trigger_flank )
      I_Contact( #ctrl.trigger_toggle )
      S_Coil( #ctrl.toggle_hulp )
   END_RUNG
   // the same network as SCL:
   IF #ctrl.trigger_flank AND NOT #ctrl.trigger_toggle THEN #ctrl.toggle_hulp := TRUE; END_IF;
END_REGION

REGION Network 3
   RUNG wire#powerrail
      Contact( #ctrl.trigger_flank )
      Contact( #ctrl.trigger_toggle )
      wire#w1
      R_Coil( #ctrl.toggle_hulp )
   END_RUNG
   RUNG wire#powerrail
      I_Contact( #ctrl.step_stop )
   END_RUNG wire#w1
   // the same network as SCL:
   IF (#ctrl.trigger_flank AND #ctrl.trigger_toggle) OR NOT #ctrl.step_stop THEN
       #ctrl.toggle_hulp := FALSE;
   END_IF;
END_REGION

REGION Network 4
   RUNG wire#powerrail
      Contact( #ctrl.toggle_hulp )
      Coil( #ctrl.trigger_toggle )
   END_RUNG
   // the same network as SCL:
   #ctrl.trigger_toggle := #ctrl.toggle_hulp;
END_REGION

REGION Network 5
   RUNG wire#powerrail
      Contact( #ctrl.auto )
      wire#w1
      Coil( #ctrl.enable_step )
   END_RUNG
   RUNG wire#powerrail
      Contact( #ctrl.onestep )
      Contact( #ctrl.trigger_flank )
   END_RUNG wire#w1
   RUNG wire#powerrail
      Contact( #ctrl.step_break )
      wire#w2
      Contact( #ctrl.break_on )
   END_RUNG wire#w1
   RUNG wire#w2
      Contact( #ctrl.trigger_flank )
   END_RUNG wire#w1
   RUNG wire#powerrail
      Contact( #ctrl.step_stop )
      Contact( #ctrl.trigger_toggle )
   END_RUNG wire#w1
   // the same network as SCL:
   #ctrl.enable_step := #ctrl.auto OR (#ctrl.onestep AND #ctrl.trigger_flank) OR (#ctrl.step_break AND (#ctrl.break_on OR #ctrl.trigger_flank)) OR (#ctrl.step_stop AND #ctrl.trigger_toggle);
END_REGION
END_FUNCTION

FUNCTION "ctrl_seq" : Void   // FC16, SCL
{ S7_Optimized_Access := 'FALSE' }
VERSION : 0.1
   VAR_INPUT
      size : Int;
   END_VAR
   VAR_IN_OUT
      sequences : "grafcet_data";
   END_VAR
   VAR_TEMP
      count : Int;
      test : "CTRL";
   END_VAR
BEGIN
   #count:=0;
   REPEAT
        #count := #count + 1;
        #sequences.MyCTRL.break_on := NOT (#sequences.Mygrafcet.actual.step[#count] AND #sequences.Mygrafcet.break.step[#count]);

   UNTIL #sequences.Mygrafcet.actual.step[#count] AND #sequences.Mygrafcet.break.step[#count] OR (#count = #size) END_REPEAT;

   #test := #sequences.MyCTRL;
   "Grafcet_modus"(#test);
   #sequences.MyCTRL := #test;

   #sequences.Mygrafcet.old := #sequences.Mygrafcet.actual;
END_FUNCTION

FUNCTION "initialisation" : Void   // FC100, SCL
{ S7_Optimized_Access := 'FALSE' }
VERSION : 0.1
   VAR_INPUT
      number : Int;
   END_VAR
   VAR_IN_OUT
      Normal_sequence : "grafcet_data";
   END_VAR
   VAR_TEMP
      lus : Int;
   END_VAR
BEGIN
   #Normal_sequence.Mygrafcet.actual.step[0] := false;
   #Normal_sequence.Mygrafcet.old.step[0] := false;

   #Normal_sequence.Mygrafcet.actual.step[1] := true;
   #Normal_sequence.Mygrafcet.old.step[1] := true;

   FOR #lus :=2  TO #number DO

       #Normal_sequence.Mygrafcet.actual.step[#lus] := false;
       #Normal_sequence.Mygrafcet.old.step[#lus] := false;

       // Statement section FOR
       ;
   END_FOR;
END_FUNCTION

// ===== PLC "PLC_1"  CPU 1516-3 PN/DP =====

VAR_GLOBAL   // PLC tag table "Default tag table"
   "start" AT %I124.0 : Bool;
   "stop" AT %I124.1 : Bool;
   "a1" AT %I124.4 : Bool;   // InsertionManueelDownward
   "a0" AT %I124.5 : Bool;
   "b0" AT %I124.6 : Bool;
   "b1" AT %I124.7 : Bool;
   "v1" AT %I125.0 : Bool;
   "c0" AT %I125.1 : Bool;
   "c1" AT %I125.2 : Bool;
   "d0" AT %I125.3 : Bool;
   "d1" AT %I125.4 : Bool;
   "v2" AT %I125.5 : Bool;
   "f1" AT %I125.6 : Bool;
   "g0" AT %I125.7 : Bool;
   "g1" AT %I126.0 : Bool;
   "j0" AT %I126.1 : Bool;
   "dm" AT %I126.2 : Bool;
   "dp" AT %I126.3 : Bool;
   "e_stop" AT %I126.4 : Bool;
   "auto_man" AT %I124.2 : Bool;
   "reset" AT %I124.3 : Bool;
   "ER" AT %Q124.0 : Bool;
   "A+" AT %Q124.1 : Bool;
   "B+" AT %Q124.2 : Bool;
   "V1+" AT %Q124.3 : Bool;
   "C+" AT %Q124.4 : Bool;
   "C-" AT %Q124.5 : Bool;
   "D+" AT %Q124.6 : Bool;
   "V2+" AT %Q124.7 : Bool;
   "E+" AT %Q125.0 : Bool;
   "F+" AT %Q125.1 : Bool;
   "G+" AT %Q125.2 : Bool;
   "H+" AT %Q125.3 : Bool;
   "I+" AT %Q125.4 : Bool;
   "J+" AT %Q125.5 : Bool;
   "K+" AT %Q125.6 : Bool;
   "FM" AT %Q125.7 : Bool;
END_VAR

TYPE "Sequence"
VERSION : 0.1
   STRUCT
      actual : "step";
      old : "step";
      break : "step";
   END_STRUCT;
END_TYPE

TYPE "step"
VERSION : 0.1
   STRUCT
      "step" : Array[0..25] of Bool;
   END_STRUCT;
END_TYPE

TYPE "CTRL"
VERSION : 0.1
   STRUCT
      emergency_stop : Bool;
      trigger : Bool;
      trigger_flank : Bool;
      trigger_toggle : Bool;
      trigger_hulp : Bool;
      enable_step : Bool;
      auto : Bool;
      onestep : Bool;
      step_stop : Bool;
      step_break : Bool;
      toggle_hulp : Bool;
      break_on : Bool;
   END_STRUCT;
END_TYPE

TYPE "grafcet_data"
VERSION : 0.1
   STRUCT
      MyCTRL : "CTRL";
      Mygrafcet : "Sequence";
   END_STRUCT;
END_TYPE

TYPE "carousel"
   STRUCT
      carousel : Array[0..7] of Int;
   END_STRUCT;
END_TYPE

DATA_BLOCK "Tafel_As_DB"   // DB1
{ S7_Optimized_Access := 'FALSE' }
VERSION : 0.1
// stored: InstanceOfName Tafel_As
"Tafel_As"
BEGIN
END_DATA_BLOCK

DATA_BLOCK "inhoud_car_tab"   // DB3
{ S7_Optimized_Access := 'TRUE' }
VERSION : 0.1
   VAR
      data : "carousel";
   END_VAR
BEGIN
END_DATA_BLOCK

FUNCTION_BLOCK "Tafel_As"   // FB1, SCL
{ S7_Optimized_Access := 'FALSE' }
VERSION : 0.1
   VAR_INPUT
      start : Bool;
      sensorA0 : Bool;
      sensorA1 : Bool;
      sensorB0 : Bool;
      sensorB1 : Bool;
      sensorC0 : Bool;
      sensorC1 : Bool;
      sensorD0 : Bool;
      sensorD1 : Bool;
      sensorF1 : Bool;
      sensorG0 : Bool;
      sensorG1 : Bool;
      sensorV1 : Bool;
      sensorV2 : Bool;
      sensorDm : Bool;
      sensorDp : Bool;
      sensorJ0 : Bool;
   END_VAR
   VAR_OUTPUT
      "CilA+" : Bool;
      "CilB+" : Bool;
      "CilC+" : Bool;
      "CilC-" : Bool;
      "CilD+" : Bool;
      "CilE+" : Bool;
      "CilF+" : Bool;
      "CilG+" : Bool;
      "CilH+" : Bool;
      "CilI+" : Bool;
      "CilK+" : Bool;
      "CilJ+" : Bool;
      "ZV1+" : Bool;
      "ZV2+" : Bool;
   END_VAR
   VAR
      "cilinderA+" : "cilinder";
      "cilinderB+" : "cilinder";
      "cilinderC+" : "cilinder";
      "cilinderC-" : "cilinder";
      "cilinderD+" : "cilinder";
      "cilinderE+" : "cilinder";
      "cilinderF+" : "cilinder";
      "cilinderG+" : "cilinder";
      "cilinderH+" : "cilinder";
      "cilinderI+" : "cilinder";
      "cilinderK+" : "cilinder";
      "cilinderJ+" : "cilinder";
      "zuigerV1+" : "cilinder";
      "zuigerV2+" : "cilinder";
      seq_as_einde_invoer : "grafcet_data";
      seq_as_draaien_invoer : "grafcet_data";
      seq_sorteringsarm_invoer : "grafcet_data";
      seq_detectiesensoren_invoer : "grafcet_data";
      seq_carousel_invoer : "grafcet_data";
      seq_plaatsen_as : "grafcet_data";
      timer300ms : TON_TIME;
      Twist_caro_as : "Twist_caro";
      test : Int;
      Schrijf_pos_caro_as : "Schrijf_pos_caro";
      timer100ms : TON_TIME;
      Lees_pos_caro_as : "Lees_pos_caro";
      positie3 : Int;
      positie6 : Int;
      positie7 : Int;
   END_VAR
BEGIN
   REGION Aanmaken grafcets
       // Statement section REGION
       "ctrl_seq"(size := 10,
                  sequences := #seq_as_einde_invoer);

       "ctrl_seq"(size := 10,
                  sequences := #seq_as_draaien_invoer);

       "ctrl_seq"(size := 10,
                  sequences := #seq_sorteringsarm_invoer);

       "ctrl_seq"(size := 10,
                  sequences := #seq_detectiesensoren_invoer);

       "ctrl_seq"(size := 10,
                  sequences := #seq_carousel_invoer);

       "ctrl_seq"(size := 10,
                  sequences := #seq_plaatsen_as);
   END_REGION

   REGION Stappen
       // Statement section REGION
       REGION Stappen grafcet carousel
           // Statement section REGION

           "Seq1-->1"(actualstep := 0,
                      nextstep := 1,
                      condition := #start,
                      Sequence := #seq_carousel_invoer);

           "Seq1-->1"(actualstep := 1,
                      nextstep := 2,
                      condition := #sensorJ0,
                      Sequence := #seq_carousel_invoer);

           "Seq1-->1"(actualstep := 2,
                      nextstep := 3,
                      condition := #seq_as_draaien_invoer.Mygrafcet.actual.step[8] AND #seq_as_einde_invoer.Mygrafcet.actual.step[9] AND #seq_sorteringsarm_invoer.Mygrafcet.actual.step[5] AND #seq_plaatsen_as.Mygrafcet.actual.step[2],
                      Sequence := #seq_carousel_invoer);

           "Seq1-->1"(actualstep := 3,
                      nextstep := 4,
                      condition := #timer300ms.Q,
                      Sequence := #seq_carousel_invoer);

           "Seq1-->1"(actualstep := 4,
                      nextstep := 5,
                      condition := #timer300ms.Q AND #sensorJ0 = FALSE,
                      Sequence := #seq_carousel_invoer);

           "Seq1-->1"(actualstep := 5,
                      nextstep := 1,
                      condition := #timer300ms.Q,
                      Sequence := #seq_carousel_invoer);

       END_REGION

       REGION Stappen grafcet as plaatsen en meten, detecteren stukken
           // Statement section REGION

           "Seq1-->1"(actualstep := 1,
                      nextstep := 2,
                      condition := #seq_carousel_invoer.Mygrafcet.actual.step[5],
                      Sequence := #seq_plaatsen_as);

           "Seq1-->1"(actualstep := 2,
                      nextstep := 1,
                      condition := #timer100ms.Q,
                      Sequence := #seq_plaatsen_as);
       END_REGION

       REGION Stappen grafcet as draaien
           // Statement section REGION

           IF #positie3 = 0 THEN
               "Seq1-->1"(actualstep := 1,
                          nextstep := 2,
                          condition := #sensorG0 AND #seq_carousel_invoer.Mygrafcet.actual.step[5],
                          Sequence := #seq_as_draaien_invoer);
           ELSE
               "Seq1-->1"(actualstep := 1,
                          nextstep := 8,
                          condition := #sensorG0 AND #seq_carousel_invoer.Mygrafcet.actual.step[5],
                          Sequence := #seq_as_draaien_invoer);
           END_IF;

           "Seq1-->1"(actualstep := 2,
                      nextstep := 3,
                      condition := #sensorG1,
                      Sequence := #seq_as_draaien_invoer);

           "Seq1-->1"(actualstep := 3,
                      nextstep := 4,
                      condition := #timer300ms.Q,
                      Sequence := #seq_as_draaien_invoer);

           "Seq1-->1"(actualstep := 4,
                      nextstep := 5,
                      condition := #sensorG0,
                      Sequence := #seq_as_draaien_invoer);

           "Seq1-->1"(actualstep := 5,
                      nextstep := 6,
                      condition := #timer300ms.Q,
                      Sequence := #seq_as_draaien_invoer);

           "Seq1-->1"(actualstep := 6,
                      nextstep := 7,
                      condition := #sensorG1,
                      Sequence := #seq_as_draaien_invoer);

           "Seq1-->1"(actualstep := 7,
                      nextstep := 8,
                      condition := #sensorG1,
                      Sequence := #seq_as_draaien_invoer);

           "Seq1-->1"(actualstep := 8,
                      nextstep := 1,
                      condition := #timer300ms.Q,
                      Sequence := #seq_as_draaien_invoer);
       END_REGION

       REGION Stappen grafset sorteringsarm
           // Statement section REGION

           IF #positie6 = 0 THEN
               "Seq1-->1"(actualstep := 1,
                          nextstep := 2,
                          condition := #sensorC0 AND #seq_carousel_invoer.Mygrafcet.actual.step[5],
                          Sequence := #seq_sorteringsarm_invoer);
           ELSE
               "Seq1-->1"(actualstep := 1,
                          nextstep := 5,
                          condition := #sensorC0 AND #seq_carousel_invoer.Mygrafcet.actual.step[5],
                          Sequence := #seq_sorteringsarm_invoer);
           END_IF;

           "Seq1-->1"(actualstep := 2,
                      nextstep := 3,
                      condition := #sensorC1,
                      Sequence := #seq_sorteringsarm_invoer);

           "Seq1-->1"(actualstep := 3,
                      nextstep := 4,
                      condition := #sensorD1,
                      Sequence := #seq_sorteringsarm_invoer);

           "Seq1-->1"(actualstep := 4,
                      nextstep := 5,
                      condition := #sensorV2,
                      Sequence := #seq_sorteringsarm_invoer);

           "Seq1-->1"(actualstep := 5,
                      nextstep := 1,
                      condition := #sensorD0,
                      Sequence := #seq_sorteringsarm_invoer);
       END_REGION

       REGION Stappen grafcet as plaatsen op lager
           // Statement section REGION

           IF #positie7 = 1 THEN
               "Seq1-->1"(actualstep := 1,
                          nextstep := 2,
                          condition := #sensorB0 AND #seq_carousel_invoer.Mygrafcet.actual.step[5],
                          Sequence := #seq_as_einde_invoer);
           ELSE
               "Seq1-->1"(actualstep := 1,
                          nextstep := 9,
                          condition := #sensorB0 AND #seq_carousel_invoer.Mygrafcet.actual.step[5],
                          Sequence := #seq_as_einde_invoer);
           END_IF;

           "Seq1-->1"(actualstep := 2,
                      nextstep := 3,
                      condition := #sensorA0,
                      Sequence := #seq_as_einde_invoer);

           "Seq1-->1"(actualstep := 3,
                      nextstep := 4,
                      condition := #sensorA1,
                      Sequence := #seq_as_einde_invoer);

           "Seq1-->1"(actualstep := 4,
                      nextstep := 5,
                      condition := #sensorV1,
                      Sequence := #seq_as_einde_invoer);

           "Seq1-->1"(actualstep := 5,
                      nextstep := 6,
                      condition := #sensorA0,
                      Sequence := #seq_as_einde_invoer);

           "Seq1-->1"(actualstep := 6,
                      nextstep := 7,
                      condition := #sensorB1,
                      Sequence := #seq_as_einde_invoer);

           "Seq1-->1"(actualstep := 7,
                      nextstep := 8,
                      condition := #sensorA1,
                      Sequence := #seq_as_einde_invoer);

           "Seq1-->1"(actualstep := 8,
                      nextstep := 9,
                      condition := #timer300ms.Q,
                      Sequence := #seq_as_einde_invoer);

           "Seq1-->1"(actualstep := 9,
                      nextstep := 1,
                      condition := #sensorA0,
                      Sequence := #seq_as_einde_invoer);
       END_REGION
   END_REGION

   REGION Uitgangen
       // Statement section REGION
       REGION Uitgang as plaatsen en meten
           // Statement section REGION

           #"cilinderE+"(AutomatischUitschuiven := #seq_plaatsen_as.Mygrafcet.actual.step[1],
                         AansturingMono => #"CilE+");


           #"cilinderF+"(AutomatischUitschuiven := #seq_plaatsen_as.Mygrafcet.actual.step[2],
                         AansturingMono => #"CilF+");

       END_REGION

       REGION Uitgangen as draaien
           // Statement section REGION
           #"cilinderH+"(AutomatischUitschuiven := #seq_as_draaien_invoer.Mygrafcet.actual.step[4] OR #seq_as_einde_invoer.Mygrafcet.actual.step[5] OR #seq_as_einde_invoer.Mygrafcet.actual.step[6] OR #seq_as_einde_invoer.Mygrafcet.actual.step[7],
                         AansturingMono => #"CilH+");

           #"cilinderG+"(AutomatischUitschuiven := #seq_as_draaien_invoer.Mygrafcet.actual.step[1] OR #seq_as_draaien_invoer.Mygrafcet.actual.step[2] OR #seq_as_draaien_invoer.Mygrafcet.actual.step[5] OR #seq_as_draaien_invoer.Mygrafcet.actual.step[6],
                         AansturingMono => #"CilG+");


           #"cilinderI+"(AutomatischUitschuiven := #seq_as_draaien_invoer.Mygrafcet.actual.step[2] OR #seq_as_draaien_invoer.Mygrafcet.actual.step[3] OR #seq_as_draaien_invoer.Mygrafcet.actual.step[4] OR #seq_as_draaien_invoer.Mygrafcet.actual.step[5],
                         AansturingMono => #"CilI+");

       END_REGION

       REGION Uitgangen as plaatsen op lager
           // Statement section REGION
           #"cilinderA+"(AutomatischUitschuiven := #seq_as_einde_invoer.Mygrafcet.actual.step[2] OR #seq_as_einde_invoer.Mygrafcet.actual.step[3] OR #seq_as_einde_invoer.Mygrafcet.actual.step[6] OR #seq_as_einde_invoer.Mygrafcet.actual.step[7],
                         AansturingMono => #"CilA+");


           #"cilinderB+"(AutomatischUitschuiven := #seq_as_einde_invoer.Mygrafcet.actual.step[5] OR #seq_as_einde_invoer.Mygrafcet.actual.step[6] OR #seq_as_einde_invoer.Mygrafcet.actual.step[7] OR #seq_as_einde_invoer.Mygrafcet.actual.step[8],
                         AansturingMono => #"CilB+");

           #"zuigerV1+"(AutomatischUitschuiven := #seq_as_einde_invoer.Mygrafcet.actual.step[3] OR #seq_as_einde_invoer.Mygrafcet.actual.step[4] OR #seq_as_einde_invoer.Mygrafcet.actual.step[5] OR #seq_as_einde_invoer.Mygrafcet.actual.step[6],
                        AansturingMono => #"ZV1+");
       END_REGION

       REGION Uitgangen sorteringsarm
           // Statement section REGION
           #"cilinderC+"(AutomatischUitschuiven := #seq_sorteringsarm_invoer.Mygrafcet.actual.step[1],
                         AansturingMono => #"CilC+");

           #"cilinderC-"(AutomatischUitschuiven := #seq_sorteringsarm_invoer.Mygrafcet.actual.step[5],
                         AansturingMono => #"CilC-");

           #"cilinderD+"(AutomatischUitschuiven := #seq_sorteringsarm_invoer.Mygrafcet.actual.step[2] OR #seq_sorteringsarm_invoer.Mygrafcet.actual.step[3],
                         AansturingMono => #"CilD+");

           #"zuigerV2+"(AutomatischUitschuiven := #seq_sorteringsarm_invoer.Mygrafcet.actual.step[3] OR #seq_sorteringsarm_invoer.Mygrafcet.actual.step[4] OR #seq_sorteringsarm_invoer.Mygrafcet.actual.step[5],
                        AansturingMono => #"ZV2+");

       END_REGION

       REGION Uitgang carousel
           // Statement section REGION
           #"cilinderK+"(AutomatischUitschuiven := #seq_carousel_invoer.Mygrafcet.actual.step[2] OR #seq_carousel_invoer.Mygrafcet.actual.step[3],
                         AansturingMono => #"CilK+");

           #"cilinderJ+"(AutomatischUitschuiven := #seq_carousel_invoer.Mygrafcet.actual.step[3] OR #seq_carousel_invoer.Mygrafcet.actual.step[4],
                         AansturingMono => #"CilJ+");

       END_REGION
   END_REGION

   REGION Lezen tabel
       // Statement section REGION
       #Lees_pos_caro_as(lees_nu := #seq_carousel_invoer.Mygrafcet.actual.step[5],
                         Welke_pos := 3,
                         tabel := "inhoud_car_tab".data,
                         inhoud_pos => #positie3);
       #Lees_pos_caro_as(lees_nu := #seq_carousel_invoer.Mygrafcet.actual.step[5],
                         Welke_pos := 6,
                         tabel := "inhoud_car_tab".data,
                         inhoud_pos => #positie6);
       #Lees_pos_caro_as(lees_nu := #seq_carousel_invoer.Mygrafcet.actual.step[5],
                         Welke_pos := 7,
                         tabel := "inhoud_car_tab".data,
                         inhoud_pos => #positie7);
   END_REGION

   REGION Schrijven tabel
       // Statement section REGION
       REGION Schrijf positie as naar tabel
           // Statement section REGION
           #Schrijf_pos_caro_as(Schrijf_nu := #timer300ms.Q AND #seq_plaatsen_as.Mygrafcet.actual.step[2] AND NOT #sensorF1,
                                Welke_pos := 2,
                                soort_onderdeel := 0,
                                teller_caro := #Twist_caro_as.teller_caro,
                                tabel := "inhoud_car_tab".data);

           #Schrijf_pos_caro_as(Schrijf_nu := #sensorF1 AND NOT #timer300ms.Q AND #seq_plaatsen_as.Mygrafcet.actual.step[2],
                                Welke_pos := 2,
                                soort_onderdeel := 1,
                                teller_caro := #Twist_caro_as.teller_caro,
                                tabel := "inhoud_car_tab".data);
       END_REGION

       REGION schrijf posities van de sensoren
           // Statement section REGION
           #Schrijf_pos_caro_as(Schrijf_nu := #seq_carousel_invoer.Mygrafcet.actual.step[5] AND #sensorDm,
                                Welke_pos := 4,
                                soort_onderdeel := 1,
                                teller_caro := #Twist_caro_as.teller_caro,
                                tabel := "inhoud_car_tab".data);

           #Schrijf_pos_caro_as(Schrijf_nu := #seq_carousel_invoer.Mygrafcet.actual.step[5] AND NOT #sensorDm,
                                Welke_pos := 4,
                                soort_onderdeel := 0,
                                teller_caro := #Twist_caro_as.teller_caro,
                                tabel := "inhoud_car_tab".data);

           #Schrijf_pos_caro_as(Schrijf_nu := #seq_carousel_invoer.Mygrafcet.actual.step[5] AND #sensorDp,         //sensorDp is hoog wanneer er metaal wordt gedetecteerd.
                                Welke_pos := 5,
                                soort_onderdeel := 1,
                                teller_caro := #Twist_caro_as.teller_caro,
                                tabel := "inhoud_car_tab".data);

           #Schrijf_pos_caro_as(Schrijf_nu := #seq_carousel_invoer.Mygrafcet.actual.step[5] AND NOT #sensorDp,
                                Welke_pos := 5,
                                soort_onderdeel := 0,
                                teller_caro := #Twist_caro_as.teller_caro,
                                tabel := "inhoud_car_tab".data);
       END_REGION
   END_REGION

   REGION Timers
       // Statement section REGION
       #timer100ms(IN := #seq_plaatsen_as.Mygrafcet.actual.step[1],
                   PT := t#100ms);

       #timer300ms(IN := #seq_plaatsen_as.Mygrafcet.actual.step[2] OR #seq_as_einde_invoer.Mygrafcet.actual.step[7] OR #seq_as_draaien_invoer.Mygrafcet.actual.step[3] OR #seq_as_draaien_invoer.Mygrafcet.actual.step[5] OR #seq_as_draaien_invoer.Mygrafcet.actual.step[7],
                   PT := t#300ms);
   END_REGION

   #Twist_caro_as(twist := #seq_carousel_invoer.Mygrafcet.actual.step[4],
                  New_pointer_caro => #test);
END_FUNCTION_BLOCK

FUNCTION_BLOCK "Lees_pos_caro"   // FB2, SCL
{ S7_Optimized_Access := 'TRUE' }
VERSION : 0.1
   VAR_INPUT
      lees_nu : Bool;
      Welke_pos : Int;
      tabel : "carousel";
      teller_caro : Int;
   END_VAR
   VAR_OUTPUT
      inhoud_pos : Int;
   END_VAR
   VAR
      Flank_lezen : R_TRIG;
   END_VAR
   VAR_TEMP
      lees_nu_RE : Bool;
   END_VAR
BEGIN
   #Flank_lezen(CLK:=#lees_nu,
                Q=>#lees_nu_RE);

   IF #lees_nu_RE THEN
       // Statement section IF
       #inhoud_pos := #tabel.carousel[(#teller_caro - #Welke_pos) MOD 8];

   END_IF;
END_FUNCTION_BLOCK

FUNCTION_BLOCK "Twist_caro"   // FB3, SCL
{ S7_Optimized_Access := 'TRUE' }
VERSION : 0.1
   VAR_INPUT
      twist : Bool;
   END_VAR
   VAR_OUTPUT
      New_pointer_caro : Int;
   END_VAR
   VAR
      teller_caro : Int := 8;
      R_TRIG_twist : R_TRIG;
   END_VAR
   VAR_TEMP
      pos_flank : Bool;
   END_VAR
BEGIN
   #R_TRIG_twist(CLK:=#twist,
                 Q=>#pos_flank);


   IF #pos_flank THEN
       #teller_caro += 1;
       #New_pointer_caro := #teller_caro MOD 8;
   END_IF;
END_FUNCTION_BLOCK

FUNCTION_BLOCK "Schrijf_pos_caro"   // FB4, SCL
{ S7_Optimized_Access := 'TRUE' }
VERSION : 0.1
   VAR_INPUT
      Schrijf_nu : Bool;
      Welke_pos : Int;
      soort_onderdeel : Int;
      teller_caro : Int;
   END_VAR
   VAR_OUTPUT
      inhoud_pos : Int;
   END_VAR
   VAR_IN_OUT
      tabel : "carousel";
   END_VAR
   VAR
      Flank_lezen : R_TRIG;
   END_VAR
   VAR_TEMP
      Schrijf_nu_RE : Bool;
   END_VAR
BEGIN
   #Flank_lezen(CLK:=#Schrijf_nu,
                Q=>#Schrijf_nu_RE);

   IF #Schrijf_nu_RE THEN
       // Statement section IF
       #tabel.carousel[(#teller_caro - #Welke_pos) MOD 8]:= #soort_onderdeel;

   END_IF;
END_FUNCTION_BLOCK

ORGANIZATION_BLOCK "Main"   // OB1, LAD, ProgramCycle
TITLE = "Main Program Sweep (Cycle)"
{ S7_Optimized_Access := 'TRUE' }
VERSION : 0.1
   VAR_INPUT
      Initial_Call : Bool;   // Initial call of this OB
      Remanence : Bool;   // =True, if remanent data are available
   END_VAR
BEGIN

REGION Network 1
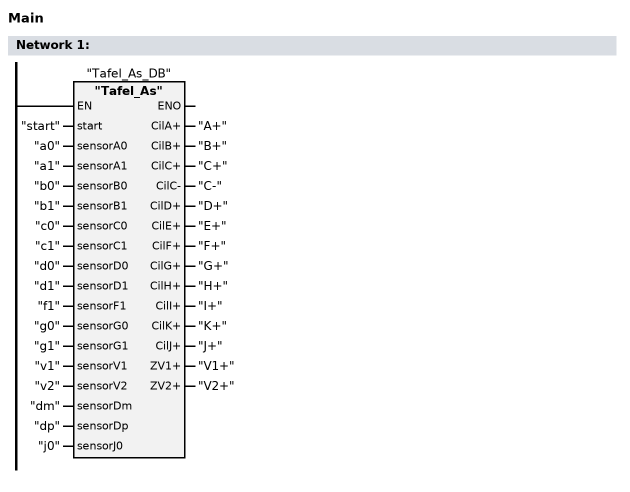
   RUNG wire#powerrail
      "Tafel_As_DB"(start := "start", sensorA0 := "a0", sensorA1 := "a1", sensorB0 := "b0", sensorB1 := "b1", sensorC0 := "c0", sensorC1 := "c1", sensorD0 := "d0", sensorD1 := "d1", sensorF1 := "f1", sensorG0 := "g0", sensorG1 := "g1", sensorV1 := "v1", sensorV2 := "v2", sensorDm := "dm", sensorDp := "dp", sensorJ0 := "j0", "CilA+" => "A+", "CilB+" => "B+", "CilC+" => "C+", "CilC-" => "C-", "CilD+" => "D+", "CilE+" => "E+", "CilF+" => "F+", "CilG+" => "G+", "CilH+" => "H+", "CilI+" => "I+", "CilK+" => "K+", "CilJ+" => "J+", "ZV1+" => "V1+", "ZV2+" => "V2+")
   END_RUNG
   // the same network as SCL:
   "Tafel_As_DB"(start := "start",   // "Tafel_As"
                 sensorA0 := "a0",
                 sensorA1 := "a1",
                 sensorB0 := "b0",
                 sensorB1 := "b1",
                 sensorC0 := "c0",
                 sensorC1 := "c1",
                 sensorD0 := "d0",
                 sensorD1 := "d1",
                 sensorF1 := "f1",
                 sensorG0 := "g0",
                 sensorG1 := "g1",
                 sensorV1 := "v1",
                 sensorV2 := "v2",
                 sensorDm := "dm",
                 sensorDp := "dp",
                 sensorJ0 := "j0",
                 "CilA+" => "A+",
                 "CilB+" => "B+",
                 "CilC+" => "C+",
                 "CilC-" => "C-",
                 "CilD+" => "D+",
                 "CilE+" => "E+",
                 "CilF+" => "F+",
                 "CilG+" => "G+",
                 "CilH+" => "H+",
                 "CilI+" => "I+",
                 "CilK+" => "K+",
                 "CilJ+" => "J+",
                 "ZV1+" => "V1+",
                 "ZV2+" => "V2+");
END_REGION
END_ORGANIZATION_BLOCK

// folder: basisclasses

FUNCTION_BLOCK "cilinder"   // FB8, FBD
{ S7_Optimized_Access := 'FALSE' }
VERSION : 0.1
   VAR_INPUT
      manueelinschuiven : Bool;
      manueeluitschuiven : Bool;   // '1' betekent uitschuiven '0' inschuiven
      AutomatischUitschuiven : Bool;
      ManAuto : Bool;   // '1' betekent Manueel '0' Automatisch
      "IL uitschuiven" : Bool;   // '1' betekent vergrendeld
      "IL inschuiven" : Bool;   // '1' betekent vergrendeld
      "Eindeloop In" : Bool;
      "Eindeloop Uit" : Bool;
      "Reset Foutmelding" : Bool;
      TeachMode : Bool;   // '1' wanneer er tijden worden ingesteld
      MargeLooptijden : Time;   // marge instellen looptijdbewaking
      "Max Aantal slagen" : Int;   // Aantal slagen voor onderhoud
      "Reset Onderhoud" : Bool;
      Noodstop : Bool;   // '0' betekent noodstop actief
   END_VAR
   VAR_OUTPUT
      AansturingMono : Bool;
      AansturingAanBist : Bool;
      AansturingUitBist : Bool;
      "Alarm Looptijd" : Bool;   // Te lang om dicht of open te schuiven
      "Alarm Interlock" : Bool;   // poging om te bedienen bij aanwezige interlock
      "Alarm Noodstop" : Bool;
      "Alarm Eindeloop" : Bool;   // wanneer elektrisch probleem op eindelopen
      "Alarm Onderhoud" : Bool;
   END_VAR
   VAR
      grafcetssturing : Bool;
      "Referentie Looptijd Inschuiven" : Time;
      "Referentie Looptijd Uitschuiven" : Time;
      "Werkelijke Looptijd Inschuiven" : Time;
      "Werkelijke Looptijd Uitschuiven" : Time;
      "Werkelijke Aantal Slagen" : Int;
      OnderhoudTeller : CTD_INT;
      SROnderhoud : Bool;
      SREindeloop : Bool;
      SRNoodstop : Bool;
      FlankManUit : Bool;
      FlankAutoUit : Bool;
      SRInterlock : Bool;
      FlankManIN : Bool;
      FlankAutoIN : Bool;
      TeachTimer : TON_TIME;
      FlankEindeUit : Bool;
      FlankEindeIn : Bool;
      RefTijdIn : Int;
      RefTijdUit : Int;
      WerkTijdIn : Int;
      WerkTijdUit : Int;
      SRLooptijd : Bool;
      FlankEindeUit1 : Bool;
      FlankEindeIn1 : Bool;
      eindeloopuitflank : Bool;
      eindeloopinflank : Bool;
      bewaaktijdeninschuiven : "bewaaktijden";
      bewaaktijdenuitschuif : "bewaaktijden";
      flankmanueelinschuiven : Bool;
      flankmanueeluitschuiven : Bool;
      movesetreset : Bool;
      PercentageSlagen : Real;
      Real_aantal : Real;
      Monosturing : Bool;
      BisturingAan : Bool;
      BisturingUit : Bool;
      FposAansturing : Bool;
      FnegAansturing : Bool;
      DINT_aantal : DInt;
   END_VAR
   VAR_TEMP
      ondergrensin : Int;
      bovengrensuit : Int;
      ondergrensuit : Int;
      vals : Bool;
      bovengrensin : Int;
   END_VAR
   VAR_TEMP   // added for the SCL form of the ladder/FBD networks
      _w1 : Bool;
      _w2 : Bool;
      _w3 : Bool;
      _w4 : Bool;
      _w5 : Bool;
   END_VAR
BEGIN

REGION Network 1: Onderhoud
   // Teller van de cilindir om na x aantal slagen onderhoud uit te voeren op de cilindir.
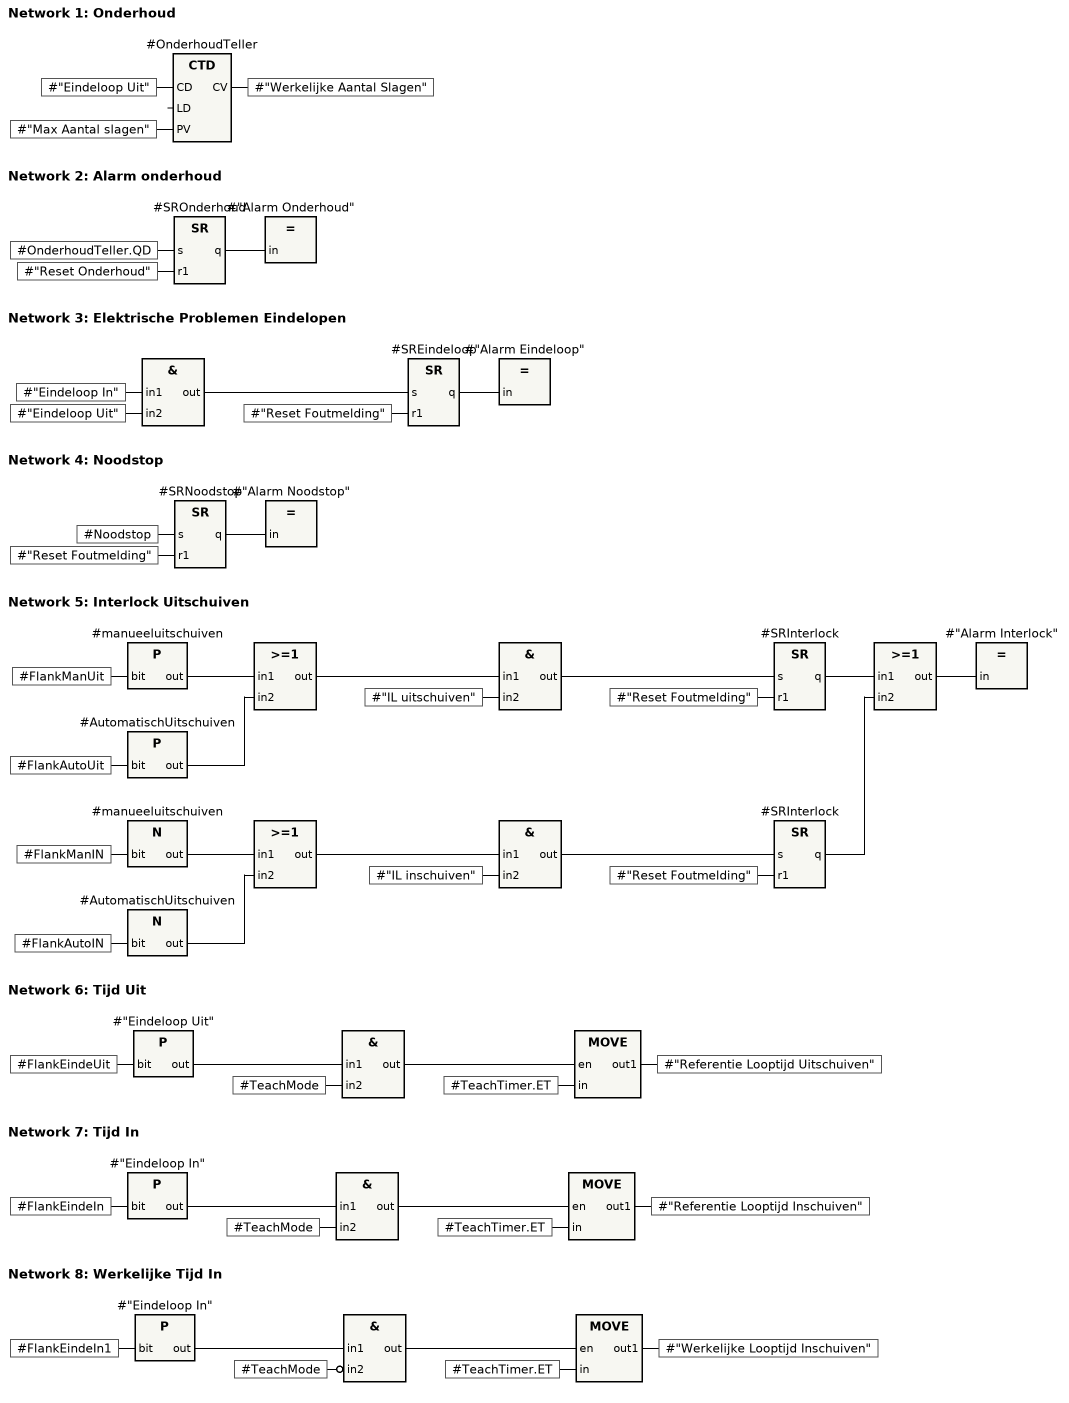
   #OnderhoudTeller(CD := #"Eindeloop Uit", PV := #"Max Aantal slagen", CV => #"Werkelijke Aantal Slagen");   // CTD
END_REGION

REGION Network 2: Alarm onderhoud
   // Weergave van wanneer de teller zijn aantal slagen heeft bereikt, kan gereset worden
   IF #OnderhoudTeller.QD THEN
       #SROnderhoud := TRUE;   // SR flip-flop
   END_IF;
   IF #"Reset Onderhoud" THEN #SROnderhoud := FALSE; END_IF;
   #"Alarm Onderhoud" := #SROnderhoud;
END_REGION

REGION Network 3: Elektrische Problemen Eindelopen
   // Beide eindelopen mogen nooit beide aanliggen, dit is fysisch niet mogelijk en is dus een elektrisch probleem
   IF #"Eindeloop In" AND #"Eindeloop Uit" THEN
       #SREindeloop := TRUE;   // SR flip-flop
   END_IF;
   IF #"Reset Foutmelding" THEN #SREindeloop := FALSE; END_IF;
   #"Alarm Eindeloop" := #SREindeloop;
END_REGION

REGION Network 4: Noodstop
   // de fysishe noodstop is nc contact
   IF #Noodstop THEN
       #SRNoodstop := TRUE;   // SR flip-flop
   END_IF;
   IF #"Reset Foutmelding" THEN #SRNoodstop := FALSE; END_IF;
   #"Alarm Noodstop" := #SRNoodstop;
END_REGION

REGION Network 5: Interlock Uitschuiven
   // Alarm voor wanneer de cilindir wordt aangestuurd maar de interlock is actief.
   #_w1 := #manueeluitschuiven AND NOT #FlankManUit;   // rising edge of #manueeluitschuiven
   #FlankManUit := #manueeluitschuiven;
   #_w2 := #AutomatischUitschuiven AND NOT #FlankAutoUit;   // rising edge of #AutomatischUitschuiven
   #FlankAutoUit := #AutomatischUitschuiven;
   IF (#_w1 OR #_w2) AND #"IL uitschuiven" THEN
       #SRInterlock := TRUE;   // SR flip-flop
   END_IF;
   IF #"Reset Foutmelding" THEN #SRInterlock := FALSE; END_IF;
   #_w3 := NOT #manueeluitschuiven AND #FlankManIN;   // falling edge of #manueeluitschuiven
   #FlankManIN := #manueeluitschuiven;
   #_w4 := NOT #AutomatischUitschuiven AND #FlankAutoIN;   // falling edge of #AutomatischUitschuiven
   #FlankAutoIN := #AutomatischUitschuiven;
   #_w5 := #SRInterlock;
   IF (#_w3 OR #_w4) AND #"IL inschuiven" THEN
       #SRInterlock := TRUE;   // SR flip-flop
   END_IF;
   IF #"Reset Foutmelding" THEN #SRInterlock := FALSE; END_IF;
   #"Alarm Interlock" := #_w5 OR #SRInterlock;
END_REGION

REGION Network 6: Tijd Uit
   // cilinder in teach mode vastleggen referentietijd uitschuiven
   #_w1 := #"Eindeloop Uit" AND NOT #FlankEindeUit;   // rising edge of #"Eindeloop Uit"
   #FlankEindeUit := #"Eindeloop Uit";
   IF #_w1 AND #TeachMode THEN #"Referentie Looptijd Uitschuiven" := #TeachTimer.ET; END_IF;
END_REGION

REGION Network 7: Tijd In
   // cilinder in teach mode vastleggen referentietijd inschuiven
   #_w1 := #"Eindeloop In" AND NOT #FlankEindeIn;   // rising edge of #"Eindeloop In"
   #FlankEindeIn := #"Eindeloop In";
   IF #_w1 AND #TeachMode THEN #"Referentie Looptijd Inschuiven" := #TeachTimer.ET; END_IF;
END_REGION

REGION Network 8: Werkelijke Tijd In
   // cilinder niet in teach mode vastleggen werkelijke tijd inschuiven
   #_w1 := #"Eindeloop In" AND NOT #FlankEindeIn1;   // rising edge of #"Eindeloop In"
   #FlankEindeIn1 := #"Eindeloop In";
   IF #_w1 AND NOT #TeachMode THEN #"Werkelijke Looptijd Inschuiven" := #TeachTimer.ET; END_IF;
END_REGION

REGION Network 9: Werkelijke Tijd Uit
   // cilinder niet in teach mode vastleggen werkelijke tijd uitschuiven
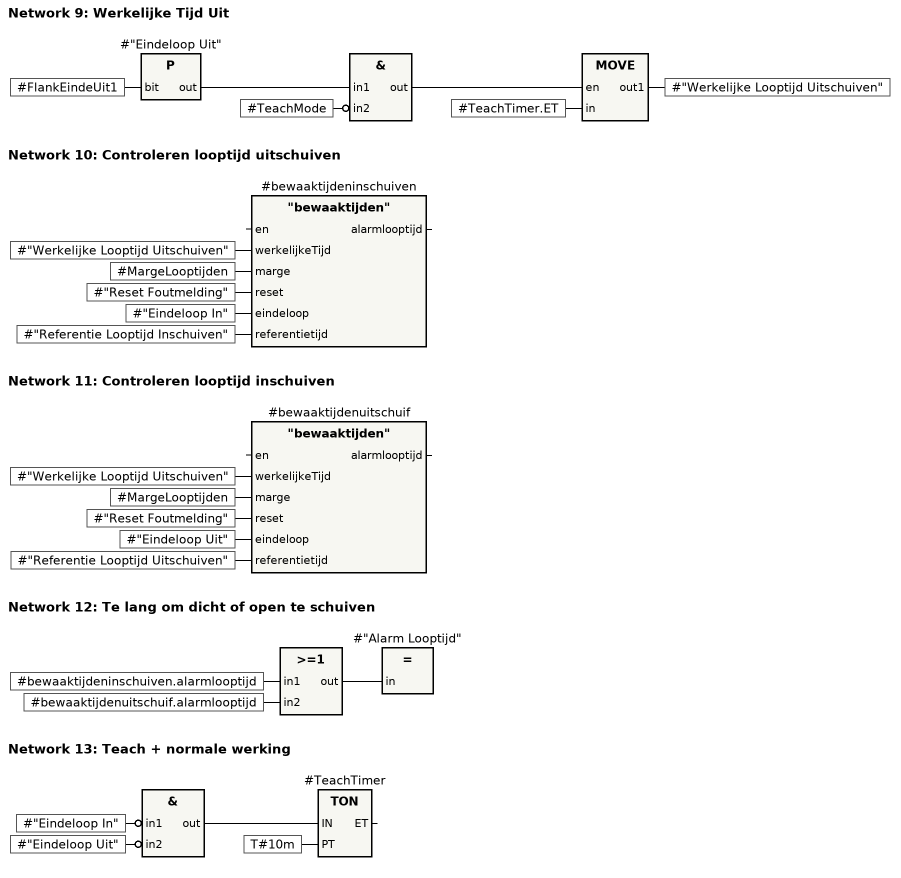
   #_w1 := #"Eindeloop Uit" AND NOT #FlankEindeUit1;   // rising edge of #"Eindeloop Uit"
   #FlankEindeUit1 := #"Eindeloop Uit";
   IF #_w1 AND NOT #TeachMode THEN #"Werkelijke Looptijd Uitschuiven" := #TeachTimer.ET; END_IF;
END_REGION

REGION Network 10: Controleren looptijd uitschuiven
   #bewaaktijdeninschuiven(werkelijkeTijd := #"Werkelijke Looptijd Uitschuiven",   // "bewaaktijden"
                           marge := #MargeLooptijden,
                           reset := #"Reset Foutmelding",
                           eindeloop := #"Eindeloop In",
                           referentietijd := #"Referentie Looptijd Inschuiven");
END_REGION

REGION Network 11: Controleren looptijd inschuiven
   #bewaaktijdenuitschuif(werkelijkeTijd := #"Werkelijke Looptijd Uitschuiven",   // "bewaaktijden"
                          marge := #MargeLooptijden,
                          reset := #"Reset Foutmelding",
                          eindeloop := #"Eindeloop Uit",
                          referentietijd := #"Referentie Looptijd Uitschuiven");
END_REGION

REGION Network 12: Te lang om dicht of open te schuiven
   #"Alarm Looptijd" := #bewaaktijdeninschuiven.alarmlooptijd OR #bewaaktijdenuitschuif.alarmlooptijd;
END_REGION

REGION Network 13: Teach + normale werking
   #TeachTimer(IN := NOT #"Eindeloop In" AND NOT #"Eindeloop Uit", PT := T#10m);   // TON
END_REGION

REGION Network 14: Sturen van de cilinder monostabiel
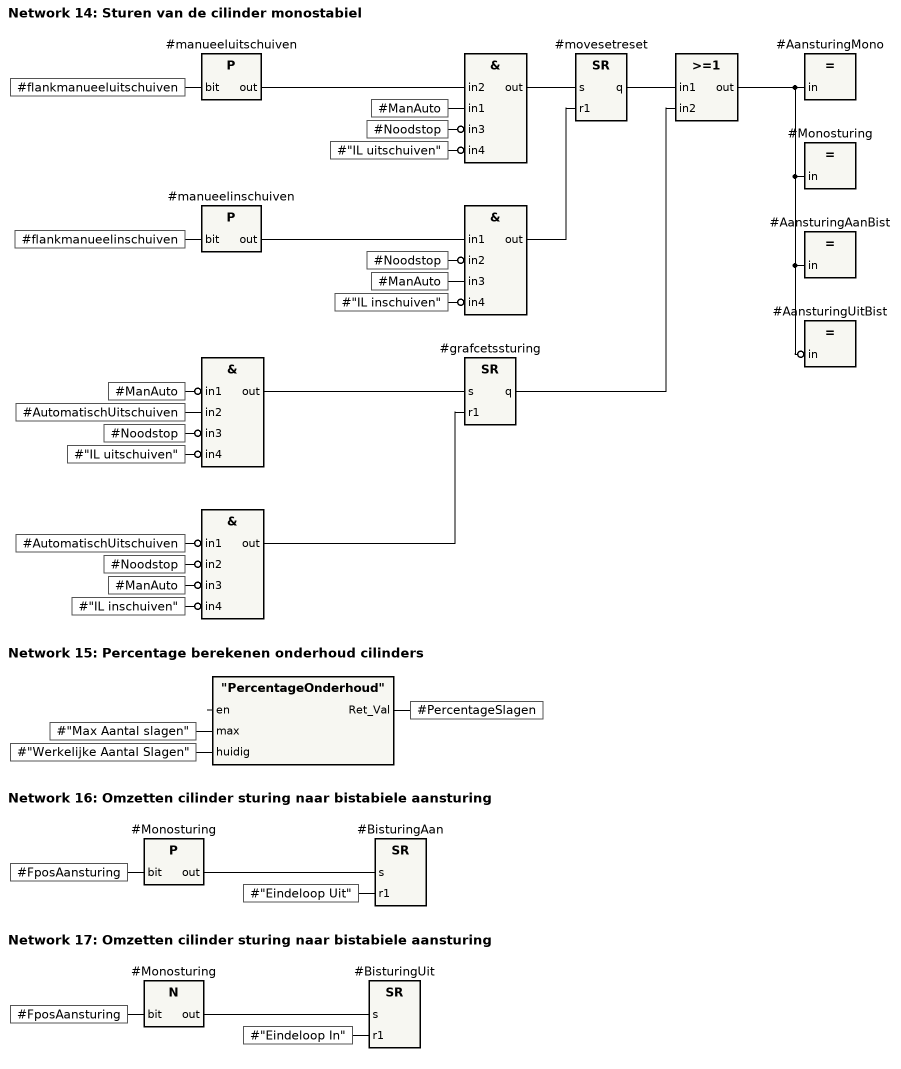
   #_w1 := #manueeluitschuiven AND NOT #flankmanueeluitschuiven;   // rising edge of #manueeluitschuiven
   #flankmanueeluitschuiven := #manueeluitschuiven;
   #_w2 := #manueelinschuiven AND NOT #flankmanueelinschuiven;   // rising edge of #manueelinschuiven
   #flankmanueelinschuiven := #manueelinschuiven;
   IF #_w1 AND #ManAuto AND NOT #Noodstop AND NOT #"IL uitschuiven" THEN
       #movesetreset := TRUE;   // SR flip-flop
   END_IF;
   IF #_w2 AND NOT #Noodstop AND #ManAuto AND NOT #"IL inschuiven" THEN #movesetreset := FALSE; END_IF;
   IF NOT #ManAuto AND #AutomatischUitschuiven AND NOT #Noodstop AND NOT #"IL uitschuiven" THEN
       #grafcetssturing := TRUE;   // SR flip-flop
   END_IF;
   IF NOT #AutomatischUitschuiven AND NOT #Noodstop AND NOT #ManAuto AND NOT #"IL inschuiven" THEN
       #grafcetssturing := FALSE;
   END_IF;
   #AansturingMono := #movesetreset OR #grafcetssturing;
   #Monosturing := #AansturingMono;
   #AansturingAanBist := #AansturingMono;
   #AansturingUitBist := NOT #AansturingMono;
END_REGION

REGION Network 15: Percentage berekenen onderhoud cilinders
   #PercentageSlagen := "PercentageOnderhoud"(max := #"Max Aantal slagen",
                           huidig := #"Werkelijke Aantal Slagen");
END_REGION

REGION Network 16: Omzetten cilinder sturing naar bistabiele aansturing
   #_w1 := #Monosturing AND NOT #FposAansturing;   // rising edge of #Monosturing
   #FposAansturing := #Monosturing;
   IF #_w1 THEN
       #BisturingAan := TRUE;   // SR flip-flop
   END_IF;
   IF #"Eindeloop Uit" THEN #BisturingAan := FALSE; END_IF;
END_REGION

REGION Network 17: Omzetten cilinder sturing naar bistabiele aansturing
   #_w1 := NOT #Monosturing AND #FposAansturing;   // falling edge of #Monosturing
   #FposAansturing := #Monosturing;
   IF #_w1 THEN
       #BisturingUit := TRUE;   // SR flip-flop
   END_IF;
   IF #"Eindeloop In" THEN #BisturingUit := FALSE; END_IF;
END_REGION
END_FUNCTION_BLOCK

FUNCTION_BLOCK "bewaaktijden"   // FB9, SCL
{ S7_Optimized_Access := 'FALSE' }
VERSION : 0.1
   VAR_INPUT
      werkelijkeTijd : Time;
      marge : Time;
      reset : Bool;
      eindeloop : Bool;
      referentietijd : Time;
   END_VAR
   VAR_OUTPUT
      alarmlooptijd : Bool;
   END_VAR
   VAR
      flankeindeloop : Bool;
   END_VAR
BEGIN
   IF ((#werkelijkeTijd > (#referentietijd + #marge)) OR (#werkelijkeTijd< (#referentietijd - #marge))) AND #eindeloop AND (NOT #flankeindeloop) THEN
       // Statement section IF
       #alarmlooptijd := TRUE;
   END_IF;
   IF #reset THEN
       // Statement section IF
       #alarmlooptijd := FALSE;
   END_IF;
   #flankeindeloop := #eindeloop;
END_FUNCTION_BLOCK

FUNCTION "PercentageOnderhoud" : Real   // FC2, SCL
{ S7_Optimized_Access := 'FALSE' }
VERSION : 0.1
   VAR_INPUT
      max : Int;
      huidig : Int;
   END_VAR
BEGIN
   #PercentageOnderhoud := INT_TO_REAL(#huidig) / INT_TO_REAL(#max) * 100;
END_FUNCTION

// folder: grafcet

FUNCTION "Seq1-->1" : Void   // FC1, SCL
{ S7_Optimized_Access := 'FALSE' }
VERSION : 0.1
   VAR_INPUT
      actualstep : Int;
      nextstep : Int;
      condition : Bool;
   END_VAR
   VAR_IN_OUT
      Sequence : "grafcet_data";
   END_VAR
BEGIN
   //Fonction permettant de passer d'une étape à une autre.


   IF #Sequence.Mygrafcet.old.step[#actualstep] AND #Sequence.MyCTRL.enable_step AND #condition THEN
       // Statement section IF
       #Sequence.Mygrafcet.actual.step[#nextstep] := true;
       #Sequence.Mygrafcet.actual.step[#actualstep] := false;

   END_IF;
END_FUNCTION

FUNCTION "Seq1-->2" : Void   // FC3, SCL
{ S7_Optimized_Access := 'FALSE' }
VERSION : 0.1
   VAR_INPUT
      actualstep : Int;
      nextstep1 : Int;
      nextstep2 : Int;
      condition : Bool;
   END_VAR
   VAR_IN_OUT
      Normal_Sequence : "grafcet_data";
   END_VAR
   VAR_TEMP
      VarConditon2 : Bool;
      VarConditon1 : Bool;
   END_VAR
BEGIN
   IF #Normal_Sequence.Mygrafcet.old.step[#actualstep] AND #Normal_Sequence.MyCTRL.enable_step AND #condition THEN
       // Statement section IF

       #Normal_Sequence.Mygrafcet.actual.step[#nextstep1] := true;
       #Normal_Sequence.Mygrafcet.actual.step[#nextstep2] := true;
       #Normal_Sequence.Mygrafcet.actual.step[#actualstep] := false;
       ;
   END_IF;
END_FUNCTION

FUNCTION "Seq2-->1" : Void   // FC4, SCL
{ S7_Optimized_Access := 'FALSE' }
VERSION : 0.1
   VAR_INPUT
      actualstep1 : Int;
      actualstep2 : Int;
      nextstep : Int;
      condition : Bool;
   END_VAR
   VAR_IN_OUT
      Normal_Sequence : "grafcet_data";
   END_VAR
BEGIN
   IF #Normal_Sequence.Mygrafcet.old.step[#actualstep1] AND #Normal_Sequence.Mygrafcet.old.step[#actualstep2] AND #Normal_Sequence.MyCTRL.enable_step AND #condition THEN
       // Statement section IF

       #Normal_Sequence.Mygrafcet.actual.step[#actualstep2] := FALSE;
       #Normal_Sequence.Mygrafcet.actual.step[#nextstep] := true;
       #Normal_Sequence.Mygrafcet.actual.step[#actualstep1] := false;
       ;
   END_IF;
END_FUNCTION

FUNCTION "Seq1--> END" : Void   // FC5, SCL
{ S7_Optimized_Access := 'FALSE' }
VERSION : 0.1
   VAR_INPUT
      actualstep : Int;
   END_VAR
   VAR_IN_OUT
      Sequence : "grafcet_data";
   END_VAR
BEGIN
   //Fonction permettant de passer d'une étape à une autre. Drain Step ( = missing next step)


   IF #Sequence.Mygrafcet.old.step[#actualstep] AND #Sequence.MyCTRL.enable_step THEN
       // Statement section IF    
       #Sequence.Mygrafcet.actual.step[#actualstep] := false;

   END_IF;
END_FUNCTION

FUNCTION "Grafcet_modus" : Void   // FC15, LAD
{ S7_Optimized_Access := 'FALSE' }
VERSION : 0.1
   VAR_IN_OUT
      ctrl : "CTRL";
   END_VAR
   VAR_TEMP   // added for the SCL form of the ladder/FBD networks
      _w1 : Bool;
   END_VAR
BEGIN

REGION Network 1
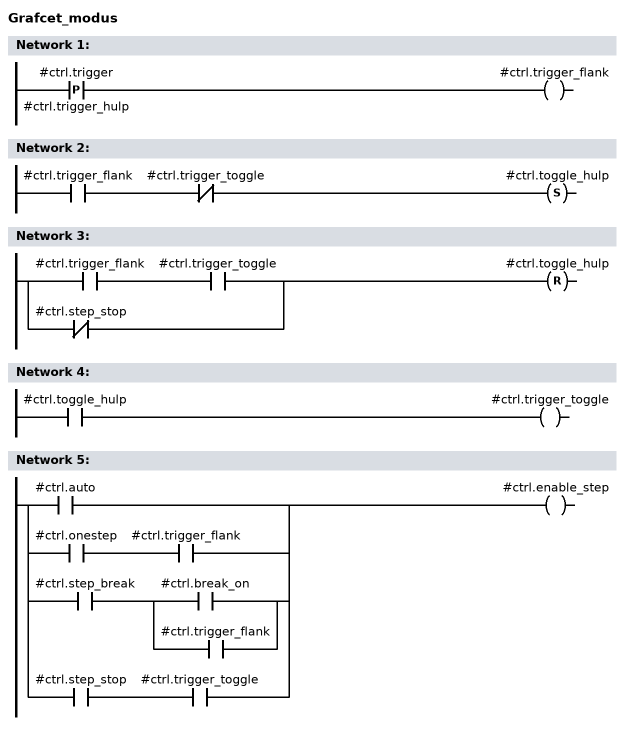
   RUNG wire#powerrail
      P_Contact(operand := #ctrl.trigger, bit := #ctrl.trigger_hulp)
      Coil( #ctrl.trigger_flank )
   END_RUNG
   // the same network as SCL:
   #_w1 := #ctrl.trigger AND NOT #ctrl.trigger_hulp;   // rising edge of #ctrl.trigger
   #ctrl.trigger_hulp := #ctrl.trigger;
   #ctrl.trigger_flank := #_w1;
END_REGION

REGION Network 2
   RUNG wire#powerrail
      Contact( #ctrl.trigger_flank )
      I_Contact( #ctrl.trigger_toggle )
      S_Coil( #ctrl.toggle_hulp )
   END_RUNG
   // the same network as SCL:
   IF #ctrl.trigger_flank AND NOT #ctrl.trigger_toggle THEN #ctrl.toggle_hulp := TRUE; END_IF;
END_REGION

REGION Network 3
   RUNG wire#powerrail
      Contact( #ctrl.trigger_flank )
      Contact( #ctrl.trigger_toggle )
      wire#w1
      R_Coil( #ctrl.toggle_hulp )
   END_RUNG
   RUNG wire#powerrail
      I_Contact( #ctrl.step_stop )
   END_RUNG wire#w1
   // the same network as SCL:
   IF (#ctrl.trigger_flank AND #ctrl.trigger_toggle) OR NOT #ctrl.step_stop THEN
       #ctrl.toggle_hulp := FALSE;
   END_IF;
END_REGION

REGION Network 4
   RUNG wire#powerrail
      Contact( #ctrl.toggle_hulp )
      Coil( #ctrl.trigger_toggle )
   END_RUNG
   // the same network as SCL:
   #ctrl.trigger_toggle := #ctrl.toggle_hulp;
END_REGION

REGION Network 5
   RUNG wire#powerrail
      Contact( #ctrl.auto )
      wire#w1
      Coil( #ctrl.enable_step )
   END_RUNG
   RUNG wire#powerrail
      Contact( #ctrl.onestep )
      Contact( #ctrl.trigger_flank )
   END_RUNG wire#w1
   RUNG wire#powerrail
      Contact( #ctrl.step_break )
      wire#w2
      Contact( #ctrl.break_on )
   END_RUNG wire#w1
   RUNG wire#w2
      Contact( #ctrl.trigger_flank )
   END_RUNG wire#w1
   RUNG wire#powerrail
      Contact( #ctrl.step_stop )
      Contact( #ctrl.trigger_toggle )
   END_RUNG wire#w1
   // the same network as SCL:
   #ctrl.enable_step := #ctrl.auto OR (#ctrl.onestep AND #ctrl.trigger_flank) OR (#ctrl.step_break AND (#ctrl.break_on OR #ctrl.trigger_flank)) OR (#ctrl.step_stop AND #ctrl.trigger_toggle);
END_REGION
END_FUNCTION

FUNCTION "ctrl_seq" : Void   // FC16, SCL
{ S7_Optimized_Access := 'FALSE' }
VERSION : 0.1
   VAR_INPUT
      size : Int;
   END_VAR
   VAR_IN_OUT
      sequences : "grafcet_data";
   END_VAR
   VAR_TEMP
      count : Int;
      test : "CTRL";
   END_VAR
BEGIN
   #count:=0;
   REPEAT
        #count := #count + 1;
        #sequences.MyCTRL.break_on := NOT (#sequences.Mygrafcet.actual.step[#count] AND #sequences.Mygrafcet.break.step[#count]);

   UNTIL #sequences.Mygrafcet.actual.step[#count] AND #sequences.Mygrafcet.break.step[#count] OR (#count = #size) END_REPEAT;

   #test := #sequences.MyCTRL;
   "Grafcet_modus"(#test);
   #sequences.MyCTRL := #test;

   #sequences.Mygrafcet.old := #sequences.Mygrafcet.actual;
END_FUNCTION

FUNCTION "initialisation" : Void   // FC100, SCL
{ S7_Optimized_Access := 'FALSE' }
VERSION : 0.1
   VAR_INPUT
      number : Int;
   END_VAR
   VAR_IN_OUT
      Normal_sequence : "grafcet_data";
   END_VAR
   VAR_TEMP
      lus : Int;
   END_VAR
BEGIN
   #Normal_sequence.Mygrafcet.actual.step[0] := false;
   #Normal_sequence.Mygrafcet.old.step[0] := false;

   #Normal_sequence.Mygrafcet.actual.step[1] := true;
   #Normal_sequence.Mygrafcet.old.step[1] := true;

   FOR #lus :=2  TO #number DO

       #Normal_sequence.Mygrafcet.actual.step[#lus] := false;
       #Normal_sequence.Mygrafcet.old.step[#lus] := false;

       // Statement section FOR
       ;
   END_FOR;
END_FUNCTION

(* ===== HMI "HMI_RT_2" =====
system functions are stored by id; their names below are inferred from use
connection "HMI_Connection_1": ETHERNET, SIMATIC S7 300/400 MPI
connection "HMI_Connection_2": ETHERNET, SMART_S7_1500_OMS

HMI tags "Default tag table"
   "Mijn_Tafel_Lager_seq_invoer_Mygrafcet_actual_step{1}" : Bool = PLC Mijn_Tafel_Lager.seq_invoer.Mygrafcet.actual.step[1] AT %DB1.DBX266.1, 1 s

screen "Screen_1" 800x480
   Rectangle "Rectangle_1" at 118,31 size 96x48
      Appearance <- "Mijn_Tafel_Lager_seq_invoer_Mygrafcet_actual_step{1}"
   Softkey "Softkey_F8" at 0,0 size 0x0
      on KeyDown: ActivateScreen("Screen_1", 0)
*)